5:	// Проверка Р2-30 и Р3-06
	IF Asda.P2_30=5 AND Asda.P3_06=3 THEN
		CNT_0:=90;
	ELSE
		IF CNT_1 = 2 THEN					// Если безушпешные 3 попытки
			Asda.E_CODE.2:=1;				// Ошибка инициализации Р2-30 или Р3-06
		ELSE		
			// Запись Р2-30=5 и Р3-06=3
			AddWriteCmd (wCmd:=wcAsda_P5_30);	// См. фукнцию AddWriteCmd	
			AddWriteCmd (wCmd:=wcAsda_P3_06);	// См. фукнцию AddWriteCmd	
			CNT_0:=10;							// Переход
		END_IF
	END_IF

10:	// Выдержка времени 1 сек
	TM_LOC (IN:=TRUE, PT:=T#1S);
	IF TM_LOC.Q THEN
		TM_LOC (IN:=FALSE);				// Сброс таймера
		CNT_0:=20;						// Переход
	END_IF

20:	// Чтение Р2-30 и Р3-06
	AddReadCmd (rCmd:=rcAsda_P2_30);	// Чтение Р2-30
	AddReadCmd (rCmd:=rcAsda_P3_06);	// Чтение Р3-06
	CNT_0:=30;							// Переход

30:	// Выдержка времени 1 сек
	TM_LOC (IN:=TRUE, PT:=T#1S);
	IF TM_LOC.Q THEN
		TM_LOC (IN:=FALSE);				// Сброс таймера
		CNT_1:=CNT_1+1;					// Увеличиваем счётчик	
		CNT_0:=5;						// Переход на начальную проверку
	END_IF

90:	// Выдержка времени 2 сек
	TM_LOC (IN:=TRUE, PT:=T#2S);
	IF TM_LOC.Q THEN
		CNT_0:=100;
	END_IF

100: // Конец 
	Asda.IsInit:=TRUE;					// Установка флага инициализации
	TM_LOC (IN:=FALSE);
	TM_DOG (IN:=FALSE);
	RESULT:=TRUE;

END_CASE

// Обнаружение ошибок
BREAK:=Asda.E_CODE <> 0;
IF BREAK THEN
	CNT_0:=100;
END_IF
END_ACTION

ACTION ST_Error_entry:

// Сброс селектора
CNT_0:=0;

// Сброс тайтера
TM_LOC (IN:=FALSE, PT:=T#2S);

// Сброс флага
RESULT:=0;

// Установить флаг ожидания сброса ошибки
Asda.WAIT_ERR:=TRUE;
END_ACTION

ACTION ST_Wait_entry:

// Включим флаг ожидания 
Asda.WAIT:=TRUE;

// Индекс сообщения
Asda.text_id:=0;
END_ACTION

ACTION ST_Servo_On_active:
CASE CNT_0 OF
0:
	// Устанавливает сигнал СБРОС и SERVO_ON на сервоприводе
	Asda.text_id:=6;					// Индекс сообщения
	AddWriteCmd (wCmd:=wcAsda_P4_07_4);	// См. функцию AddWriteCmd
	CNT_0:=10;							// Переход

10:	// Задержка 3 сек
	TM_LOC (IN:=TRUE, PT:=T#3S);
	IF TM_LOC.Q THEN
		TM_LOC (IN:=FALSE);			// Сброс таймера
		CNT_0:=20;					// Переход
	END_IF

20:	// Сбрасываем сигнал СБРОС при включенном SERVO_ON
	AddWriteCmd (wCmd:=wcAsda_P4_07_2);	// См. функцию AddWriteCmd
	CNT_0:=30;							// Переход

30:	// Задержка 1 сек
	TM_LOC (IN:=TRUE, PT:=T#1S);
	IF TM_LOC.Q THEN
		TM_LOC (IN:=FALSE);			// Сброс таймера
		CNT_0:=100;					// Переход
	END_IF

100: // Конец
	Asda.IsServo_ON:=TRUE;
	RESULT:=TRUE;

END_CASE
END_ACTION

ACTION ST_Parking_active:

CASE CNT_0 OF
	
0:	// Сообщение о движении в реперную точку
	IF Asda.IsServo_ON THEN
		Asda.text_id:=11;					// Индекс сообщения
		AddWriteCmd (wCmd:=wcAsda_Parking);	// Запуск

		CNT_0:=10;
	ELSE
		CNT_0:=100;
	END_IF
	
10:	// Ожидание 1 сек пока Р5-07 станет отличным от 20013 (Выполняется программа: PR#13 - парковка
	TM_LOC (IN:=TRUE, PT:=T#1S);
	IF TM_LOC.Q THEN
		TM_LOC (IN:=FALSE);
		CNT_0:=20;
	END_IF

20: // Ждём пока значение Р5-07 станет равно 20013 - значение окончания HOMING
	IF Asda.P5_07 = 20013 THEN
		CNT_0:=100;
	END_IF

100: // Завершение
	TM_LOC (IN:=FALSE);
	TM_DOG (IN:=FALSE);
	RESULT:=TRUE;

END_CASE

// Обнаружение предупреждения WARN (концевики в основном)
IF Asda.P0_46.10 THEN
	Asda.E_CODE.1:=1;		// WARN ()
END_IF

// Обнаруживаем ошибку АВАРИЯ СЕРВОПРИВОДА 
IF Asda.P0_46.6 THEN
	Asda.E_CODE.0:=1;		// ALRM (Авария привода)
END_IF

// Сторожевой таймер
TM_DOG (IN:=TRUE, PT:=tm_parking);
IF TM_DOG.Q THEN
	Asda.E_CODE.3:=1;		// Превышено время операции Homing
END_IF

// Ошибку блокировки игнорируем, так как будем использовать парковку
// при обработке падения темпераруры (Asda.Block) в рабочем режиме
BREAK:=Asda.E_CODE <> 0;
IF BREAK THEN 
	CNT_0:=100;
END_IF
END_ACTION

ACTION ST_Cont_entry:


// Переходим на ожидание
IF OP = OP_END THEN
    PROC:=PR_WAIT;
END_IF;
END_ACTION

ACTION ST_Stop_active:

// Экстренный останов
CASE CNT_0 OF
	
0:	// Подаём сигнал экстренного СТОП
	AddWriteCmd (wCmd:=wcAsda_Stop); 
	CNT_0:=10;
	
10:	// Небольшая задержка
	TM_LOC (IN:=TRUE, PT:=T#1S);
	IF TM_LOC.Q THEN
		TM_LOC (IN:=FALSE);
		CNT_0:=100;
	END_IF

100: // Конец
	RESULT:=TRUE;	

END_CASE
END_ACTION

ACTION ST_PR_Init_active:
CASE CNT OF

0:	// Проверка нинциализации
	IF Asda.P2_30=5 AND Asda.P3_06=3 THEN
		OP:=OP_NO;
	ELSE
		OP:=OP_INIT;
	END_IF

	CNT:=10;

10:	// Установка параметров
	OP:=OP_PARAMS;
	CNT:=100;
	
100: // Конец
	OP:=OP_END;
	
END_CASE
END_ACTION

ACTION Init_entry:

// Сброс селектора
CNT:=0;

// Начальная процедура - ожидание
PROC:=PR_WAIT;

// Сброс операции
OP:=OP_NO;

Asda.IsHoming:=FALSE;
Asda.IsInit:=FALSE;
Asda.IsServo_ON:=FALSE;
Asda.Pusk:=FALSE;
//Asda.Block:=TRUE;
Asda.WAIT:=FALSE;
Asda.WAIT_ERR:=FALSE;
Asda.WAIT_WORK:=FALSE;
Asda.P2_30:=0;
Asda.P3_06:=0;
Asda.E_CODE:=0;
Asda.text_id:=12;	// Ожидание соединения

// Проверка сохраненной ранее структуры W_Period: TPeriod
IF NOT IsRegValid (ADR (REG_W)) THEN
	REG_W:=REG_DEF;
END_IF
END_ACTION

ACTION ST_OFF_active:

CASE CNT OF
	
0:	// Инициализация сервопривода
	OP:=OP_INIT;
	CNT:=10;

10:	// Отключение сервопривода 
	OP:=OP_SERVO_OFF;
	CNT:=20;
	
20:	// Конец
	OP:=OP_END;

END_CASE
END_ACTION

ACTION ST_Stop_entry:

// Сброс селектора
CNT_0:=0;

// Сброс таймера
TM_LOC (IN:=FALSE, PT:=T#2S);

// Сброс флага
RESULT:=FALSE;

// Индекс сообщения
Asda.text_id:=7;
END_ACTION

ACTION ST_Pulsing_active:
CASE CNT_0 OF
	
0: 	// Начало
	Asda.text_id:=3;			// Индекс сообщения
	Asda.WAIT_WORK:=TRUE;		// Флаг состояния работы
	CNT_0:=10;
	
10:	// Запись команды на пульсирование
	AddWriteCmd (wCmd:=wcAsda_Working);
	CNT_0:=20;			// Переход
	
20:	// Ждём 1 сек пока значение Р5-07 изменится
	TM_LOC (IN:=TRUE, PT:=T#1S);
	IF TM_LOC.Q THEN
		TM_LOC (IN:=FALSE);
		CNT_0:=30;
	END_IF

30:

	// ЗДЕСЬ ИДЁТ ОСНОВНАЯ РАБОТА
	
	IF NOT Asda.Pusk THEN
		// Выход при автоматическом режиме
		CNT_0:=100;
	END_IF

100: // Выход

	TM_LOC (IN:=FALSE);
	TM_DOG (IN:=FALSE);
	Asda.WAIT_WORK:=FALSE;		// Флаг состояния работы
	RESULT:=TRUE;

END_CASE

// Обнаружение ошибок
IF Asda.P0_46.10 THEN
	Asda.E_CODE.1:=1;		// WARN ()
END_IF

IF Asda.P0_46.6 THEN
	Asda.E_CODE.0:=1;		// ALRM (Авария привода)
END_IF

IF Asda.E_CODE <> 0 THEN
	BREAK:=TRUE;
END_IF
	
IF BREAK THEN
	CNT_0:=100;
END_IF
END_ACTION

ACTION ST_Wait_exit:

// Выключим флаг ожидания 
Asda.WAIT:=FALSE;

// Сброс селектора
CNT:=0;

// Сброс операции
OP:=OP_NO;
END_ACTION

ACTION ST_Empty_exit:
// Внутренний селектор
CNT_0:=0;
CNT_1:=0;

// Внутренние таймеры
TM_LOC (IN:=FALSE, PT:=T#1S);
TM_DOG (IN:=FALSE, PT:=T#1S);

// Сброс флага
RESULT:=FALSE;

// Сброс прерывания
BREAK:=FALSE;
END_ACTION

ACTION ST_Params_active:

CASE CNT_0 OF

0:	// Установка индекса сообщения параметров
	Asda.text_id:=9;
	CNT_0:=10;
	
10:	// Установка параметров сервопривода
	Asda.SelButton:=sbPeriod;		// Параметры периода Asda
	AsdaSetPeriod ();

	CNT_0:=90;

90:	// Выдержка времени 2 сек
	TM_LOC (IN:=TRUE, PT:=T#2S);
	IF TM_LOC.Q THEN
		CNT_0:=100;
	END_IF

100: // Конец 
	TM_LOC (IN:=FALSE);
	TM_DOG (IN:=FALSE);
	RESULT:=TRUE;
	
END_CASE
END_ACTION

ACTION ST_FIRST_active:
CASE CNT OF

0:	// Включение сервопривода (попутно с сбросом аварии)
	OP:=OP_SERVO_ON;
	CNT:=20;			// Переход 
	
20:	// Установка параметров
	OP:=OP_PARAMS;
	CNT:=30;
	
30:	// Homing
	OP:=OP_HOMING;
	CNT:=40;
	
40:	// Конец
	OP:=OP_END;

END_CASE
END_ACTION

ACTION ST_WORK_active:

CASE CNT OF
0:	// Включение пульсирования
	OP:=OP_PULSING;
	CNT:=10;

10:	// Возвращение в реперную точку
	OP:=OP_PARKING;
	CNT:=20;	
	
20:	// Конец
	OP:=OP_END;

	
END_CASE
END_ACTION

ACTION ST_Wait_active:


// Проверяемна наличие Connect
IF Asda.Connect THEN

	IF NOT Asda.IsInit THEN
		// Инициализация
		PROC:=PR_INIT;
		FIRST:=TRUE;
		RESULT:=TRUE;
		RETURN;
	END_IF

	// Ожидание снятия блокировки (при достижении температуры)		
	IF NOT Asda.Block THEN

		// Включаем сервопривод через Servo_ON
		IF NOT Asda.IsServo_ON THEN			
			PROC:=PR_FIRST;
			RESULT:=TRUE;

		ELSIF Asda.Pusk THEN
			PROC:=PR_WORK;
			RESULT:=TRUE;
		
		END_IF

	// Появление блокировки (при снижении температуры)
	ELSE
		// Отключаем сервопривод через Servo_OFF
		IF Asda.IsServo_ON THEN
			// Инициализация, затем отключение сервопривода 
			PROC:=PR_OFF;
			RESULT:=TRUE;
		END_IF

	END_IF
END_IF
END_ACTION

ACTION ST_RESET_active:
// Процедура сброса, например после ошибки

CASE CNT OF
	
0:	// Homing
	OP:=OP_HOMING;
	CNT:=10;

10:	// Конец
	OP:=OP_END;
	
END_CASE
END_ACTION

ACTION ST_Error_active:

CASE CNT_0 OF
0:	// Ожидаем появления сигнала "СБРОС АВАРИИ"

	Asda.text_id:=10;			// Обработка ошибки
	IF ALARM_RESET THEN
		CNT_0:=10;
	END_IF

10:	// Действуем в зависимости от возникшей ошибки
	// - сигнал ALRM
	IF Asda.E_CODE.0 THEN	
		PROC:=PR_AVAR;			//	Переход на обработку аварии 	

	// - сигнал WARN	
	ELSIF Asda.E_CODE.1 THEN
		PROC:=PR_RESET;			//	Переход на Homing 	

	// - Ошибка инициализации Р2-30 или Р3-06	
	ELSIF Asda.E_CODE.2 THEN
		PROC:=PR_FIRST;			// Переход на инициализацию		
	
	// - Превышено время операции HOMING	
	ELSIF Asda.E_CODE.3 THEN
		PROC:=PR_RESET;			// Переход на Homing
	
	// - Превышено время операции отладки	
	ELSIF Asda.E_CODE.5 THEN
		PROC:=PR_RESET;			// Переход на Homing
	
	// Тестовая ошибка
	ELSIF Asda.E_CODE.6 THEN
		PROC:=PR_WAIT;			// Переход на Ожидание

	// Неизвестная ошибка
	ELSE
		PROC:=PR_WAIT;
	END_IF
	
	CNT_0:=20;					// Переход на ожидание сброса аварии

20:	// Сброс аварии
	Asda.E_CODE:=0;
	CNT_0:=30;

30: // Ожидание пропадания сигнала SBROS_AVARII
	IF NOT ALARM_RESET THEN
		CNT_0:=100;
	END_IF

100: // Конец
	RESULT:=TRUE;

END_CASE
END_ACTION

ACTION ST_Error_exit:

// Сброс операции
OP:=OP_NO;

// Сброс главного селектора
CNT:=0;

// Сбросить флаг ожидания сброса ошибки
Asda.WAIT_ERR:=FALSE;
END_ACTION

END_PROGRAM

// Device/Application/SRC/AddWriteCmd
PROGRAM AddWriteCmd
VAR_INPUT
	wCmd	: TWriteCmd;
END_VAR

VAR
	WR_CMDS		: ARRAY [0..11] OF WORD:=[5, 3, 0, 1, 2, 3, 0, 10, 13, 1000, 14, 15];	// Слова для команд сервопривода
	CH_CMDS		: ARRAY [0..1] OF WORD:=[0, 1];
	CH_UST		: INT;

END_VAR

// В зависимости от команды ...
CASE wcmd OF
	
	//=====================================================================================
	// КОМАНДЫ ПЕРВОНАЧАЛЬНОЙ ИНИЦИАЛИЗАЦИИ
	//=====================================================================================
	wcAsda_P5_30	: QueuePushReg (ADR (COM1_PRG.WR_REGS), ADR_ASDA, 16#023C, ADR (WR_CMDS[0]), 1);	// Параметр  Р2-30 -> 5 (отключение записи в EEPROM) - 5 в старшем байте!
	wcAsda_P3_06	: QueuePushReg (ADR (COM1_PRG.WR_REGS), ADR_ASDA, 16#030C, ADR (WR_CMDS[1]), 1);	// Параметр  Р3-06 -> 3 (способ управления дискретными входами) - 3 в старшем байте!
	wcAsda_P4_07_1	: QueuePushReg (ADR (COM1_PRG.WR_REGS), ADR_ASDA, 16#040E, ADR (WR_CMDS[2]), 1);	// Запись 00 в Р4-07 (servo_off)
	wcAsda_P4_07_2	: QueuePushReg (ADR (COM1_PRG.WR_REGS), ADR_ASDA, 16#040E, ADR (WR_CMDS[3]), 1);	// Запись 01 в Р4-07 (servo_on)
	wcAsda_P4_07_3	: QueuePushReg (ADR (COM1_PRG.WR_REGS), ADR_ASDA, 16#040E, ADR (WR_CMDS[4]), 1);	// Запись 10 в Р4-07 (сброс ошибок и выключенние servo_off)
	wcAsda_P4_07_4	: QueuePushReg (ADR (COM1_PRG.WR_REGS), ADR_ASDA, 16#040E, ADR (WR_CMDS[5]), 1);	// Запись 11 в Р4-07 (сброс ошибок с включенным servo_on)	
	//=====================================================================================
	// КОМАНДЫ УПРАВЛЕНИЯ ASDA
	//=====================================================================================
	wcAsda_Homing	: QueuePushReg (ADR (COM1_PRG.WR_REGS), ADR_ASDA, 16#050E, ADR (WR_CMDS[6]), 1);	// Команда HOMING - запись в Р5-07 числа 0
	wcAsda_Working	: QueuePushReg (ADR (COM1_PRG.WR_REGS), ADR_ASDA, 16#050E, ADR (WR_CMDS[7]), 1);	// Команда WORKING - запись в Р5-07 числа 10
	wcAsda_Parking	: QueuePushReg (ADR (COM1_PRG.WR_REGS), ADR_ASDA, 16#050E, ADR (WR_CMDS[8]), 1);	// Команда PARKING - запись в Р5-07 числа 13
	wcAsda_Stop		: QueuePushReg (ADR (COM1_PRG.WR_REGS), ADR_ASDA, 16#050E, ADR (WR_CMDS[9]), 1);	// КОМАНДА "СТОП" - запись в Р5-07 числа 1000
	wcAsda_Forward	: QueuePushReg (ADR (COM1_PRG.WR_REGS), ADR_ASDA, 16#050E, ADR (WR_CMDS[10]), 1);	// Команда вперёд - запись в Р5-07 числа 14
	wcAsda_Backward	: QueuePushReg (ADR (COM1_PRG.WR_REGS), ADR_ASDA, 16#050E, ADR (WR_CMDS[11]), 1);	// Команда назад - запись в Р5-07 числа 15
	//=====================================================================================
	// КОМАНДЫ ЧИЛЛЕРА
	//=====================================================================================
	wcChiller_Ust:
		CH_UST :=REAL_TO_INT (REG_W.T_CHIL * 10.0);
		QueuePushReg (ADR (COM3_PRG.WR_REGS), ADR_CHILLER, 11, ADR (CH_UST), 1);						// Запись уставки Чиллера

	wcChiller_Start	: QueuePushReg (ADR (COM3_PRG.WR_REGS), ADR_CHILLER, 12, ADR (CH_CMDS[1]), 1);		// Старт Чиллера
	wcChiller_Stop	: QueuePushReg (ADR (COM3_PRG.WR_REGS), ADR_CHILLER, 12, ADR (CH_CMDS[0]), 1);		// Стоп Чиллера
	
END_CASE

END_PROGRAM

// Device/Application/SRC/AddReadCmd
PROGRAM AddReadCmd
VAR_INPUT
	rCmd	: TReadCmd;
END_VAR

VAR
END_VAR


// В зависимости от команды 
CASE rCmd OF
	//=====================================================================================
	// КОМАНДЫ ДЛЯ ПЕРВОНАЧАЛЬНОЙ ИНИЦИАЛИЗАЦИИ ASDA_A2
	//=====================================================================================
	rcAsda_P2_30	: QueuePushReg (ADR (COM1_PRG.RD_REGS), ADR_ASDA, 16#023C, ADR (Asda.P2_30), 1); 			// Чтение Р2-30 (отключение записи в EEPROM, д.б.= 5)
	rcAsda_P3_06	: QueuePushReg (ADR (COM1_PRG.RD_REGS), ADR_ASDA, 16#030C, ADR (Asda.P3_06), 1); 			// Чтение Р3-06 (способ управления дискретными входами, д.б.= 3)
	
	
END_CASE

END_PROGRAM

// Device/Application/SRC/IsRegValid
FUNCTION IsRegValid : BOOL
VAR_INPUT
	pr : POINTER TO TReg;
	
END_VAR
VAR
	I: INT;
END_VAR

IsRegValid:=FALSE;

// Температуры
// Проверка температур
FOR I:=0 TO NUM_TEMPS-1 DO
	IF (pr^.TEMPS[I] < 0) OR (pr^.TEMPS[I] > T_CRITICALS[I]) THEN
		RETURN;
	END_IF
END_FOR

// Температура чиллера
IF (pr^.T_CHIL < 0) OR (pr^.T_CHIL > T_CHIL_CRITICAL) THEN
	RETURN;
END_IF

// Частота колебаний
IF pr^.Freq < FREQ_MIN OR pr^.Freq > FREQ_MAX THEN
	RETURN;
END_IF 

// Смещение 1-го полупериода
IF pr^.Period.Offsets[0] < (REP_MM + 0.3) OR pr^.Period.Offsets[0] > (WORK_SIZE + REP_MM - 0.3) THEN
	RETURN;
END_IF

// Смещение 2-го полупериода
IF pr^.Period.Offsets[1] < (REP_MM + 0.3) OR pr^.Period.Offsets[1] > (WORK_SIZE + REP_MM - 0.3) THEN
	RETURN;
END_IF

// Проценты полупериодов
IF pr^.Period.Per_FirstHP < ASDA_HP_MIN OR pr^.Period.Per_FirstHP > ASDA_HP_MAX THEN
	RETURN;
END_IF

// Проценты импульсов
IF pr^.Period.Per_Pulses[0] < ASDA_PULSE_MIN OR pr^.Period.Per_Pulses[0] > ASDA_PULSE_MAX THEN
	RETURN;
END_IF

IF pr^.Period.Per_Pulses[1] < ASDA_PULSE_MIN OR pr^.Period.Per_Pulses[1] > ASDA_PULSE_MAX THEN
	RETURN;
END_IF

// Проценты уровня
IF pr^.Period.Per_Levels[0] < ASDA_LEVEL_MIN OR pr^.Period.Per_Levels[0] > ASDA_LEVEL_MAX THEN
	RETURN;
END_IF

IF pr^.Period.Per_Levels[1] < ASDA_LEVEL_MIN OR pr^.Period.Per_Levels[1] > ASDA_LEVEL_MAX THEN
	RETURN;
END_IF

// Скорость заготовки
IF pr^.Speed < SPEED_MIN OR pr^.Speed >= SPEED_MAX THEN
	RETURN;
END_IF

// Длина заготовки
IF pr^.Length < LEN_MIN OR pr^.Length > LEN_MAX THEN
	RETURN;
END_IF

// Производительность
IF pr^.Qm < QM_MIN OR pr^.Qm > QM_MAX THEN
	RETURN;
END_IF

IsRegValid:=TRUE;

END_FUNCTION

// Device/Application/SRC/AsdaSetPeriod
PROGRAM AsdaSetPeriod
VAR
	dRep		: DINT;
	wSpeeds		: ARRAY [0..1] OF WORD;			// обороты в мин
	wAccs		: ARRAY [0..3] OF WORD;			// обороты в мин
	wDels		: ARRAY [0..1] OF WORD;			// милисекунды
	dOffsets	: ARRAY [0..1] OF DINT;
	dist		: REAL;
	tPeriod		: REAL;			
	tHalfs		: ARRAY [0..1] OF REAL;
	tPulses		: ARRAY [0..1] OF REAL;
	tLevels		: ARRAY [0..1] OF REAL;
	tAccs		: ARRAY [0..1] OF REAL;
	midSpeeds	: ARRAY [0..1] OF REAL;
	vSpeeds		: ARRAY [0..1] OF REAL;
END_VAR


CASE Asda.SelButton OF

sbPeriod:	// УСТАНОВКА ПАРАМЕТРОВ ПЕРИОДА

	// 1. Сначала записать положение реперной точки P6-01, адрес 16х0602
	dRep:=REAL_TO_DINT (REP_MM * PUU_PER_MM);
	QueuePushReg (ADR (COM1_PRG.WR_REGS), ADR_ASDA, 16#0602, ADR (dRep), 2);			// Р6-01 Положение реперной точки

	// 2. Запись перемещения 1-го полупериода, т.к. оно используется при вычислении следующих параметров
	dOffsets[0]:=REAL_TO_DINT (REG_W.Period.Offsets[0] * PUU_PER_MM);
	QueuePushReg (ADR (COM1_PRG.WR_REGS), ADR_ASDA, 16#062A, ADR (dOffsets[0]), 2);	// Р6-21 Смещение 1-го полупериода рабочее
	QueuePushReg (ADR (COM1_PRG.WR_REGS), ADR_ASDA, 16#063A, ADR (dOffsets[0]), 2);	// Р6-29 Смещение 1-го полупериода для ШАГА позиционирования 14 (ручное перемещение)

	// Запись перемещения 2-го полупериода, т.к. оно используется при вычислении следующих параметров
	dOffsets[1]:=REAL_TO_DINT (REG_W.Period.Offsets[1] * PUU_PER_MM);
	QueuePushReg (ADR (COM1_PRG.WR_REGS), ADR_ASDA, 16#062E, ADR (dOffsets[1]), 2);	// Р6-23 Смещение 2-го полупериода
	QueuePushReg (ADR (COM1_PRG.WR_REGS), ADR_ASDA, 16#063E, ADR (dOffsets[1]), 2);	// Р6-31 Смещение 2-го полупериода для шага позиционирования 15 (ручное перемещение)

	// Время периода в секундах
	tPeriod:= 1 / REG_W.Freq;
	
	// Времена полупериодов в секундах
	tHalfs[0]:=tPeriod * REG_W.Period.Per_FirstHP / 100;
	tHalfs[1]:=tPeriod - tHalfs[0];
	
	// Времена импульсов в секундах
	tPulses[0]:=tHalfs[0] * REG_W.Period.Per_Pulses[0] / 100;
	tPulses[1]:=tHalfs[1] * REG_W.Period.Per_Pulses[1] / 100;
	
	// Фронты полупериодов (импульсов) в секундах - Длина импульса минус длина уровня, делённая на 2
	tAccs[0]:=tPulses[0] * (100 - REG_W.Period.Per_Levels[0]) / 200;
	tAccs[1]:=tPulses[1] * (100 - REG_W.Period.Per_Levels[1]) / 200;
	
	// Уровни полупериодов
	tLevels[0]:=tPulses[0] * REG_W.Period.Per_Levels[0] / 100;
	tLevels[1]:=tPulses[1] * REG_W.Period.Per_Levels[1] / 100;
	
	// Пройденный путь в мм
	dist:=ABS (REG_W.Period.Offsets[0] - REG_W.Period.Offsets[1]);
	
	// Средние скорости в мм/сек
	midSpeeds[0]:=dist / tPulses[0];
	midSpeeds[1]:=dist / tPulses[1];
	
	// Расчётные скорости в мм/сек
	vSpeeds[0]:=midSpeeds[0] * (2 * tAccs[0] + tLevels[0]) / (tAccs[0] + tLevels[0]);
	vSpeeds[1]:=midSpeeds[1] * (2 * tAccs[1] + tLevels[1]) / (tAccs[1] + tLevels[1]);
		
	// Пересчёт скорости, данные - l оборот => 5 мм перемещения
	// 5 мм/сек = 1 об/сек =>
	wSpeeds[0]:=REAL_TO_WORD (vSpeeds[0] * 60 * 10 / 5);	// Получили в об/мин (Нужно умножить на 10, т.к. в сервоприводе единица измерения скорости 0.1 об/мин)
	wSpeeds[1]:=REAL_TO_WORD (vSpeeds[1] * 60 * 10 / 5);	// Получили в об/мин

	// Пересчёт фронт и спада относительно скорости wSpeeds[0]
	wAccs[0]:=REAL_TO_WORD (tAccs[0] * 3000 * 1000 / wSpeeds[0]);	
	wAccs[1]:=REAL_TO_WORD (tAccs[0] * 3000 * 1000 / wSpeeds[0]);
	wAccs[2]:=REAL_TO_WORD (tAccs[1] * 3000 * 1000 / wSpeeds[1]);
	wAccs[3]:=REAL_TO_WORD (tAccs[1] * 3000 * 1000 / wSpeeds[1]);
	
	// Задержки в миллисекундах
	wDels[0]:=REAL_TO_WORD ((tHalfs[0] - tPulses[0]) * 1000.0);
	wDels[1]:=REAL_TO_WORD ((tHalfs[1] - tPulses[1]) * 1000.0);

	// Запись	
	QueuePushReg (ADR (COM1_PRG.WR_REGS), ADR_ASDA, 16#0528, ADR (wAccs[0]), 1);		// Р5-20 Фронт 1-го полупериода
	QueuePushReg (ADR (COM1_PRG.WR_REGS), ADR_ASDA, 16#052A, ADR (wAccs[1]), 1);		// Р5-21 Спад 1-го полупериода 
	QueuePushReg (ADR (COM1_PRG.WR_REGS), ADR_ASDA, 16#052C, ADR (wAccs[2]), 1);		// Р5-22 Фронт 2-го полупериода
	QueuePushReg (ADR (COM1_PRG.WR_REGS), ADR_ASDA, 16#052E, ADR (wAccs[3]), 1);		// Р5-23 Спад 2-го полупериода 

	QueuePushReg (ADR (COM1_PRG.WR_REGS), ADR_ASDA, 16#0578, ADR (wSpeeds[0]), 1);		// Р5-60 Скорость 1-го полупериода
	QueuePushReg (ADR (COM1_PRG.WR_REGS), ADR_ASDA, 16#057A, ADR (wSpeeds[1]), 1);		// Р5-61 Скорость 2-го полупериода 

	QueuePushReg (ADR (COM1_PRG.WR_REGS), ADR_ASDA, 16#0550, ADR (wDels[0]), 1);		// Р5-40 Задержка 1-го полупериода
	QueuePushReg (ADR (COM1_PRG.WR_REGS), ADR_ASDA, 16#0552, ADR (wDels[1]), 1);		// Р5-41 Задержка 2-го полупериода

// Команда Homing
sbHoming: AddWriteCmd (wCmd:=wcAsda_Homing);
	
// Движение вперёд
sbForward: AddWriteCmd (wCmd:=wcAsda_Forward);

// Движение назад
sbBackward: AddWriteCmd (wCmd:=wcAsda_Backward);

// Парковка
sbParking: AddWriteCmd (wCmd:=wcAsda_Parking);

// Работа (пульсирование)
sbWorking: AddWriteCmd (wCmd:=wcAsda_Working);
	
END_CASE

Asda.SelButton:=sbNo;
Asda.bCmd:=FALSE;

END_PROGRAM

// Device/Application/SRC_AUX/SWAP_BYTES
FUNCTION SWAP_BYTES : WORD
VAR_INPUT
	wValue : WORD;
END_VAR
VAR
END_VAR


SWAP_BYTES := SHL (wValue, 8) OR SHR (wValue, 8);

END_FUNCTION

// Device/Application/SRC/SET_FRAME_INDEX_EX
FUNCTION SET_FRAME_INDEX_EX : BYTE
VAR_INPUT
	Index : BYTE;
END_VAR
VAR
END_VAR
VAR // added by the converter: edge detectors and wires of the graphical bodies
    _w1 : ANY;
END_VAR

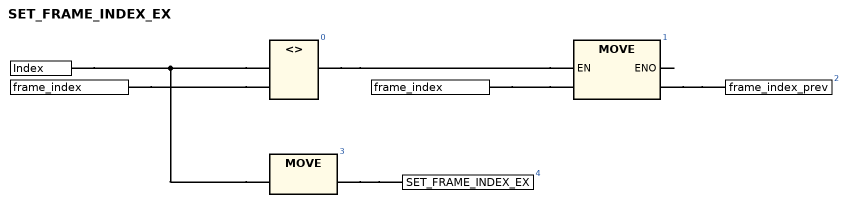
IF Index <> frame_index THEN _w1 := frame_index; END_IF
frame_index_prev := _w1;
SET_FRAME_INDEX_EX := Index;

END_FUNCTION

// Device/Application/SRC_AUX/BYTES_FROM_DINT
FUNCTION BYTES_FROM_DINT : BOOL
VAR_INPUT
	pBytes	: POINTER TO BYTE;
	iDint	: DINT;
END_VAR
VAR
	pB		: POINTER TO BYTE;
END_VAR

BYTES_FROM_DINT:=TRUE;

pB:=ADR(iDint);

pBytes[0]:=pB[1];
pBytes[1]:=pB[0];
pBytes[2]:=pB[3];
pBytes[3]:=pB[2];

END_FUNCTION

// Device/Application/SRC/MERGE_RGB
FUNCTION MERGE_RGB : DWORD
VAR_INPUT
	clR	: BYTE;
	clG	: BYTE;
	clB	: BYTE;
END_VAR
VAR
END_VAR

MERGE_RGB:=BYTE_TO_DWORD(255);
MERGE_RGB:=SHL(MERGE_RGB,8);
MERGE_RGB:=MERGE_RGB OR BYTE_TO_DWORD(clR);
MERGE_RGB:=SHL(MERGE_RGB,8);
MERGE_RGB:=MERGE_RGB OR BYTE_TO_DWORD(clG);
MERGE_RGB:=SHL(MERGE_RGB,8);
MERGE_RGB:=MERGE_RGB OR BYTE_TO_DWORD(clB);

END_FUNCTION

// Device/Application/SRC_FILE/WRITE_OPTIONS
FUNCTION WRITE_OPTIONS : BOOL
VAR_INPUT
	Show	: BOOL;
END_VAR
VAR
	hFile	: SysFile.RTS_IEC_HANDLE;	
	Result	: SysFile.RTS_IEC_RESULT;
	rSize	: __XWORD;
	wrBytes	: __XWORD;
	
END_VAR

WRITE_OPTIONS:=FALSE;
// Создаём новый файл
hFile:=SysFileOpen (OPTIONSFILE,SysFile.AM_WRITE, ADR (Result));
IF Result <> 0 THEN
	RETURN;
END_IF

rSize:=SIZEOF (TSetts);

wrBytes:=SysFileWrite(hFile, ADR (Setts), rSize, ADR (Result));
IF (Result=0) AND (wrBytes=rSize) THEN
	WRITE_OPTIONS:=TRUE;
END_IF

SysFileClose (hFile);

END_FUNCTION

// Device/Application/SRC_AUX/HiWord
FUNCTION HiWord : WORD
VAR_INPUT
	dValue	: DINT;
END_VAR	
VAR
	pW		: POINTER TO WORD;
END_VAR

pW:= ADR (dValue);
HiWord:=pW[1];

END_FUNCTION

// Device/Application/SRC_FILE/READ_OPTIONS
FUNCTION READ_OPTIONS : BOOL
VAR
	hFile	: SysFile.RTS_IEC_HANDLE;	
	Result	: SysFile.RTS_IEC_RESULT;
	fSize	: __XWORD;
	rSize	: __XWORD;
	rdBytes	: __XWORD;
	rdSetts	: TSetts;
	
END_VAR

READ_OPTIONS:=FALSE;

rSize:=SIZEOF(TSetts);

hFile:=SysFileOpen (OPTIONSFILE, SysFile.AM_READ, ADR (Result));
IF Result <> 0 THEN
	RETURN;
END_IF

//  Файл существует, проверяем размер файла
fSize:=SysFileGetSizeByHandle (hFile, ADR (Result));
IF Result <> 0 OR fSize <> rSize THEN
	SysFileClose(hFile);
	RETURN;	
END_IF

rdBytes:=SysFileRead(hFile, ADR (rdSetts), rSize, ADR (Result));	
IF Result = 0 AND rdBytes = rSize THEN
	Setts:=rdSetts;
	READ_OPTIONS:=TRUE;
END_IF

SysFileClose(hFile);

END_FUNCTION

// Device/Application/SRC_AUX/LoWord
FUNCTION LoWord : WORD
VAR_INPUT
	dValue	: DINT;
END_VAR
VAR
	pW		: POINTER TO WORD;
END_VAR

pW:= ADR (dValue);
LoWord:=pW[0];

END_FUNCTION

// Device/Application/SRC_AUX/LoByte
FUNCTION LoByte : BYTE
VAR_INPUT
	W	: WORD;
END_VAR
VAR
END_VAR

LoByte:=WORD_TO_BYTE (W AND 16#FF);

END_FUNCTION

// Device/Application/SRC_AUX/HiByte
FUNCTION HiByte : BYTE
VAR_INPUT
	W : WORD;
END_VAR
VAR
END_VAR

HiByte:= WORD_TO_BYTE (SHR (W, 8) AND 16#FF);

END_FUNCTION

// Device/Application/SRC_AUX/BYTES_FROM_INT
FUNCTION BYTES_FROM_INT : BOOL
VAR_INPUT
	pBytes	: POINTER TO BYTE;
	vInt	: INT;
END_VAR
VAR
	pB		: POINTER TO BYTE;
END_VAR

BYTES_FROM_INT:=TRUE;

pB:=ADR(vInt);
pBytes[0]:=pB[1];
pBytes[1]:=pB[0];

END_FUNCTION

// Device/Application/Visu/VIS_SETTS_2
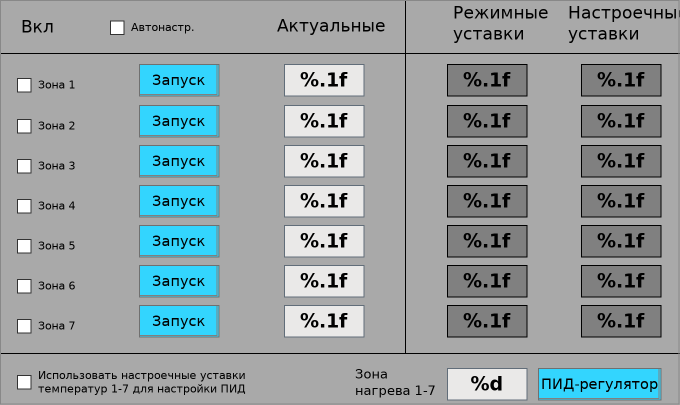
VISUALIZATION VIS_SETTS_2  // 680x405
    Checkbox (15,64 120x42), "Зона 1", variable: Nagrev.T_Enables.0
    Checkbox (15,105 120x42), "Зона 2", variable: Nagrev.T_Enables.1
    Checkbox (15,145 120x42), "Зона 3", variable: Nagrev.T_Enables.2
    Checkbox (15,185 120x42), "Зона 4", variable: Nagrev.T_Enables.3
    Checkbox (15,225 120x42), "Зона 5", variable: Nagrev.T_Enables.4
    Checkbox (15,265 120x42), "Зона 6", variable: Nagrev.T_Enables.5
    Checkbox (15,305 120x42), "Зона 7", variable: Nagrev.T_Enables.6
    Label (18,15 63x24), "Вкл"
    Button (139,64 80x32), "Запуск", colour toggle: Nagrev.Auto_IN.0, input disabled if: NOT AutoPIDActivate
        OnMouseClick: execute { Nagrev.Auto_OUT.0:=TRUE; }
    Button (139,105 80x32), "Запуск", colour toggle: Nagrev.Auto_IN.1, input disabled if: NOT AutoPIDActivate
        OnMouseClick: execute { Nagrev.Auto_OUT.1:=TRUE; }
    Button (139,145 80x32), "Запуск", colour toggle: Nagrev.Auto_IN.2, input disabled if: NOT AutoPIDActivate
        OnMouseClick: execute { Nagrev.Auto_OUT.2:=TRUE; }
    Button (139,185 80x32), "Запуск", colour toggle: Nagrev.Auto_IN.3, input disabled if: NOT AutoPIDActivate
        OnMouseClick: execute { Nagrev.Auto_OUT.3:=TRUE; }
    Button (139,225 80x32), "Запуск", colour toggle: Nagrev.Auto_IN.4, input disabled if: NOT AutoPIDActivate
        OnMouseClick: execute { Nagrev.Auto_OUT.4:=TRUE; }
    Button (139,265 80x32), "Запуск", colour toggle: Nagrev.Auto_IN.5, input disabled if: NOT AutoPIDActivate
        OnMouseClick: execute { Nagrev.Auto_OUT.5:=TRUE; }
    Button (139,305 80x32), "Запуск", colour toggle: Nagrev.Auto_IN.6, input disabled if: NOT AutoPIDActivate
        OnMouseClick: execute { Nagrev.Auto_OUT.6:=TRUE; }
    Checkbox (15,361 312x42), "Использовать настроечные уставки температур 1-7 для настройки ПИД", variable: zd_selector
    RoundedRectangle (447,64 80x32), "%.1f", text variable: REG_W.TEMPS[0], colour toggle: NOT zd_selector
    RoundedRectangle (447,105 80x32), "%.1f", text variable: REG_W.TEMPS[1], colour toggle: NOT zd_selector
    RoundedRectangle (447,145 80x32), "%.1f", text variable: REG_W.TEMPS[2], colour toggle: NOT zd_selector
    RoundedRectangle (447,185 80x32), "%.1f", text variable: REG_W.TEMPS[3], colour toggle: NOT zd_selector
    RoundedRectangle (447,225 80x32), "%.1f", text variable: REG_W.TEMPS[4], colour toggle: NOT zd_selector
    RoundedRectangle (447,265 80x32), "%.1f", text variable: REG_W.TEMPS[5], colour toggle: NOT zd_selector
    RoundedRectangle (447,305 80x32), "%.1f", text variable: REG_W.TEMPS[6], colour toggle: NOT zd_selector
    Label (450,1 107x49), "Режимные уставки"
    RoundedRectangle (581,64 80x32), "%.1f", text variable: zd_temps[0], colour toggle: zd_selector
        OnMouseClick: write the text variable via VisuDialogs.Numpad, min T_MINS_ZAD[6], max T_MAXS_ZAD[6], title "ТЕМПЕРАТУРА 7 ЗОНЫ"
    RoundedRectangle (581,105 80x32), "%.1f", text variable: zd_temps[1], colour toggle: zd_selector
        OnMouseClick: write the text variable via VisuDialogs.Numpad, min T_MINS_ZAD[0], max T_MAXS_ZAD[0]
    RoundedRectangle (581,145 80x32), "%.1f", text variable: zd_temps[2], colour toggle: zd_selector
        OnMouseClick: write the text variable via VisuDialogs.Numpad, min T_MINS_ZAD[0], max T_MAXS_ZAD[0]
    RoundedRectangle (581,185 80x32), "%.1f", text variable: zd_temps[3], colour toggle: zd_selector
        OnMouseClick: write the text variable via VisuDialogs.Numpad, min T_MINS_ZAD[0], max T_MAXS_ZAD[0]
    RoundedRectangle (581,225 80x32), "%.1f", text variable: zd_temps[4], colour toggle: zd_selector
        OnMouseClick: write the text variable via VisuDialogs.Numpad, min T_MINS_ZAD[0], max T_MAXS_ZAD[0]
    RoundedRectangle (581,265 80x32), "%.1f", text variable: zd_temps[5], colour toggle: zd_selector
        OnMouseClick: write the text variable via VisuDialogs.Numpad, min T_MINS_ZAD[0], max T_MAXS_ZAD[0]
    RoundedRectangle (581,305 80x32), "%.1f", text variable: zd_temps[6], colour toggle: zd_selector
        OnMouseClick: write the text variable via VisuDialogs.Numpad, min T_MINS_ZAD[0], max T_MAXS_ZAD[0]
    Label (565,1 127x47), "Настроечные уставки"
    RoundedRectangle (284,64 80x32), "%.1f", text variable: Nagrev.T_Actuals[0], colour variable: Nagrev.FillColors[0]
        p3450524324: Nagrev.FrameColors[0]
    RoundedRectangle (284,105 80x32), "%.1f", text variable: Nagrev.T_Actuals[1], colour variable: Nagrev.FillColors[1]
        p3450524324: Nagrev.FrameColors[1]
    RoundedRectangle (284,145 80x32), "%.1f", text variable: Nagrev.T_Actuals[2], colour variable: Nagrev.FillColors[2]
        p3450524324: Nagrev.FrameColors[2]
    RoundedRectangle (284,185 80x32), "%.1f", text variable: Nagrev.T_Actuals[3], colour variable: Nagrev.FillColors[3]
        p3450524324: Nagrev.FrameColors[3]
    RoundedRectangle (284,225 80x32), "%.1f", text variable: Nagrev.T_Actuals[4], colour variable: Nagrev.FillColors[4]
        p3450524324: Nagrev.FrameColors[4]
    RoundedRectangle (284,265 80x32), "%.1f", text variable: Nagrev.T_Actuals[5], colour variable: Nagrev.FillColors[5]
        p3450524324: Nagrev.FrameColors[5]
    RoundedRectangle (284,305 80x32), "%.1f", text variable: Nagrev.T_Actuals[6], colour variable: Nagrev.FillColors[6]
        p3450524324: Nagrev.FrameColors[6]
    Label (274,14 123x32), "Актуальные"
    Label (352,365 91x40), "Зона нагрева 1-7"
    Button (538,368 123x32), "ПИД-регулятор"
        OnMouseClick:  Dialog=DlgPids, Parameters={bDialogVar: b_dialog}, Selected={1: }, OpenModal=True, OpenCentered=True
    RoundedRectangle (447,368 80x32), "%d", text variable: Dvp.zone_index
        OnMouseClick: write the text variable via VisuDialogs.Numpad, min 1, max 7, title "Введите зону нагрева 1-7"
    Line (405,0) (405,353)
    Line (0,353) (680,353)
    Checkbox (108,9 140x37), "Автонастр.", variable: AutoPIDActivate
    Line (0,53) (680,53)
END_VISUALIZATION

// Device/Application/Visu/Main_Panel
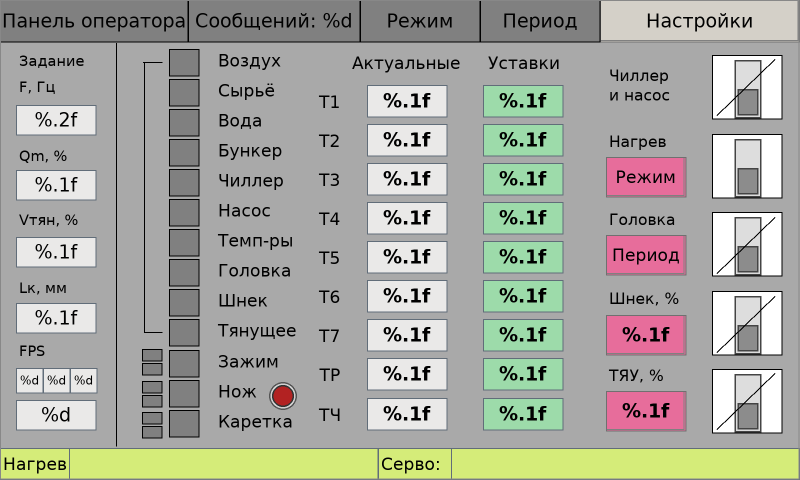
VISUALIZATION Main_Panel  // 800x480
    Rectangle (0,448 80x32), "Нагрев:"
    Frame (118,43 692x442), frame switch variable: frame_index
        shows VIS_OPERATOR()
        shows VIS_MSGS()
        shows VIS_REG()
        shows VIS_PERIOD()
        shows VIS_REG()
    Label (16,77 48x25), "F, Гц"
    RoundedRectangle (16,170 80x30), "%.1f", text variable: Shnek.Qm
    Label (16,146 77x27), "Qm, %"
    Label (16,210 92x26), "Vтян, %"
    RoundedRectangle (16,237 80x30), "%.1f", text variable: Pulling.Speed
    Label (16,278 59x25), "Lк, мм"
    RoundedRectangle (16,303 80x30), "%.1f", text variable: REG_W.Length
    RoundedRectangle (16,105 80x30), "%.2f", text variable: REG_W.Freq
    Label (16,51 79x20), "Задание"
    Line (116,43) (116,446)
    Rectangle (0,0 188x42), "Панель оператора", colour toggle: frame_index=0
        OnMouseClick: execute { SET_FRAME_INDEX (0); }
    Rectangle (188,0 172x42), "Сообщений: %d", text variable: alarm_count, colour toggle: frame_index=1
        OnMouseClick: execute { SET_FRAME_INDEX (1); }
    Button (600,0 200x42), "Настройки"
        OnMouseClick:  Assign=Setts_Panel, Type=Assignment
    Rectangle (69,448 309x32), text list: 'DvpTextList', text index: Nagrev.text_id
    Rectangle (378,448 80x32), "Серво:"
    Rectangle (451,448 349x32), text list: 'AsdaTextList', text index: Asda.text_id
    RoundedRectangle (16,400 80x30), "%d", text variable: FPS_FULL
    Label (16,341 59x25), "FPS"
    RoundedRectangle (16,368 27x25), "%d", text variable: COM1_PRG.FPS
    RoundedRectangle (43,368 27x25), "%d", text variable: COM2_PRG.FPS
    RoundedRectangle (70,368 27x25), "%d", text variable: COM3_PRG.FPS
    Rectangle (360,0 120x42), "Режим", colour toggle: frame_index=2
        OnMouseClick: execute { SET_FRAME_INDEX (2); }
    Rectangle (480,0 120x42), "Период", colour toggle: frame_index=3
        OnMouseClick: execute { SET_FRAME_INDEX (3); }
END_VISUALIZATION

// Device/Application/Visu/DlgConfirm
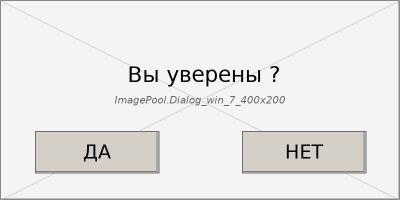
VISUALIZATION DlgConfirm  // 400x200
VAR_IN_OUT
	bDialogVar	: BOOL;
END_VAR
    Image (0,0 400x200), image: ImagePool.Dialog_win_7_400x200
    Button (35,131 124x42), "ДА"
        OnMouseClick:  Dialog=DlgConfirm, Result=OK, NumpadKeypadSet=True
        OnMouseClick: execute { bDialogVar:=TRUE; }
    Button (242,131 124x42), "НЕТ"
        OnMouseClick:  Dialog=DlgConfirm, Result=Cancel, NumpadKeypadSet=True
    Label (80,55 248x39), "Вы уверены ?"
END_VISUALIZATION

// Device/Application/Visu/Panel_Reg
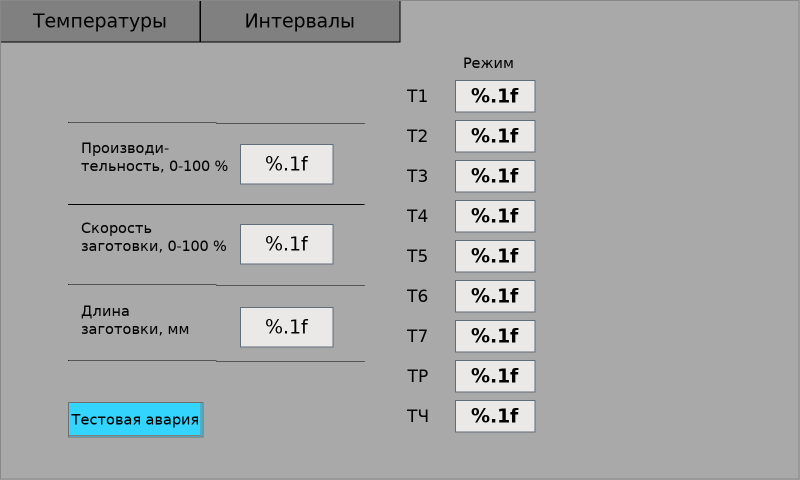
VISUALIZATION Panel_Reg  // 800x480
    Frame (6,47 734x398), frame switch variable: frame_index_reg
        shows VIS_REG()
        shows VIS_PERIOD()
    Rectangle (0,0 200x42), "Температуры", colour toggle: frame_index_reg=0
        OnMouseClick: execute { frame_index_reg:=0; }
    Rectangle (200,0 200x42), "Интервалы", colour toggle: frame_index_reg=1
        OnMouseClick: execute { frame_index_reg:=1; }
END_VISUALIZATION

// Device/Application/Visu/VIS_MSGS
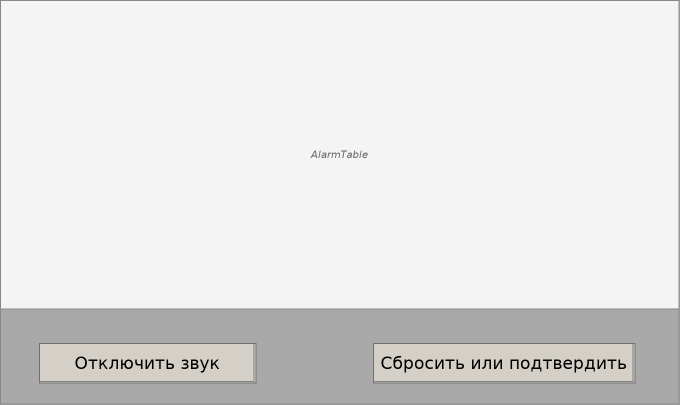
VISUALIZATION VIS_MSGS  // 680x405
VAR_IN_OUT
END_VAR
VAR
	bAckSel : BOOL;
	bAckVisible : BOOL;
	bHistory : BOOL;
	bFreezeScrlPos : BOOL;
END_VAR
    AlarmTable (0,0 679x309)
        Column[0]: ColumnTitle=Изоб
        Column[1]: ColumnTitle=Сообщение
        p1521930926: __All
        p1663851261: __All
        p428520879: bAckSel
        p2607059081: bAckVisible
        p3266827225: bHistory
        p3894972949: bFreezeScrlPos
    Button (39,343 217x40), "Отключить звук", colour toggle: ALARM_ZVUK AND NOT Setts.otkl_alarm_zvuk
        OnMouseClick: execute { ALARM_ZVUK:=FALSE; }
    Button (373,343 262x40), "Сбросить или подтвердить", colour toggle: ALARM_RESET
        toggle bAckVisible
        OnMouseClick: execute { ALARM_RESET:=TRUE; }
END_VISUALIZATION

// Device/Application/Visu/Setts_Panel
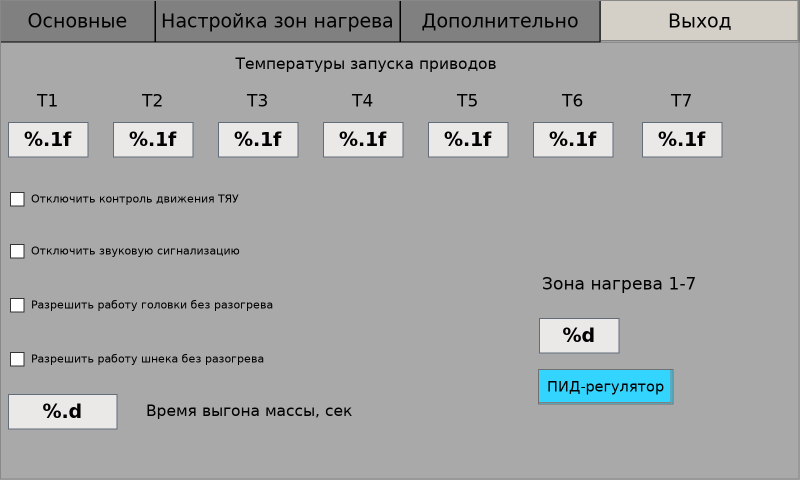
VISUALIZATION Setts_Panel  // 800x480
    Button (600,0 200x42), "Выход"
        OnMouseClick:  Assign=Main_Panel, Type=Assignment
    Rectangle (0,0 155x42), "Основные", colour toggle: frame_index_setts=0
        OnMouseClick: execute { frame_index_setts:=0; }
    Rectangle (155,0 245x42), "Настройка зон нагрева", colour toggle: frame_index_setts=1
        OnMouseClick: execute { frame_index_setts:=1; }
    Frame (0,43 793x430), frame switch variable: frame_index_setts
        shows VIS_SETTS_1()
        shows VIS_SETTS_2()
        shows VIS_SETTS_3()
    Rectangle (400,0 200x42), "Дополнительно", colour toggle: frame_index_setts=2
        OnMouseClick: execute { frame_index_setts:=2; }
END_VISUALIZATION

// Device/Application/Visu/VIS_REG
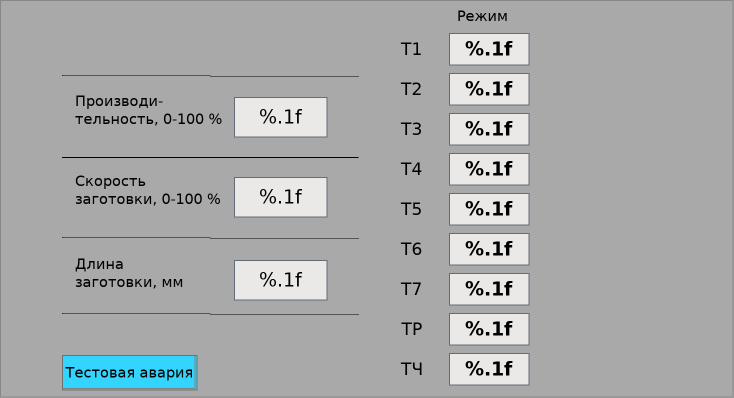
VISUALIZATION VIS_REG  // 734x398
    Line (62,313) (358,314)
    Line (62,237) (358,238)
    Line (62,157) (358,157)
    Line (62,75) (358,76)
    Label (72,91 162x53), "Производи- тельность, 0-100 %"
    Label (72,171 167x50), "Скорость заготовки, 0-100 %"
    RoundedRectangle (234,177 93x40), "%.1f", text variable: REG_W.Speed
        OnMouseClick: write the text variable via VisuDialogs.Numpad, min SPEED_MIN, max SPEED_MAX, title "Скорость заготовки, мм/сек"
    Label (72,254 126x53), "Длина заготовки, мм"
    RoundedRectangle (234,260 93x40), "%.1f", text variable: REG_W.Length
        OnMouseClick: write the text variable via VisuDialogs.Numpad, min LEN_MIN, max LEN_MAX, title "Длина заготовки, мм"
    RoundedRectangle (449,33 80x32), "%.1f", text variable: REG_W.TEMPS[0]
        OnMouseClick: write the text variable via VisuDialogs.Numpad, min T_MINS_ZAD[0], max T_MAXS_ZAD[0], title "ТЕМПЕРАТУРА 1 ЗОНЫ"
    Label (392,33 40x32), "T1"
    RoundedRectangle (449,73 80x32), "%.1f", text variable: REG_W.TEMPS[1]
        OnMouseClick: write the text variable via VisuDialogs.Numpad, min T_MINS_ZAD[1], max T_MAXS_ZAD[1], title "ТЕМПЕРАТУРА 2 ЗОНЫ"
    Label (392,73 40x32), "T2"
    RoundedRectangle (449,113 80x32), "%.1f", text variable: REG_W.TEMPS[2]
        OnMouseClick: write the text variable via VisuDialogs.Numpad, min T_MINS_ZAD[2], max T_MAXS_ZAD[2], title "ТЕМПЕРАТУРА3 ЗОНЫ"
    Label (392,113 40x32), "T3"
    RoundedRectangle (449,153 80x32), "%.1f", text variable: REG_W.TEMPS[3]
        OnMouseClick: write the text variable via VisuDialogs.Numpad, min T_MINS_ZAD[3], max T_MAXS_ZAD[3], title "ТЕМПЕРАТУРА 4 ЗОНЫ"
    Label (392,153 40x32), "T4"
    RoundedRectangle (449,193 80x32), "%.1f", text variable: REG_W.TEMPS[4]
        OnMouseClick: write the text variable via VisuDialogs.Numpad, min T_MINS_ZAD[4], max T_MAXS_ZAD[4], title "ТЕМПЕРАТУРА 5 ЗОНЫ"
    Label (392,193 40x32), "T5"
    RoundedRectangle (449,233 80x32), "%.1f", text variable: REG_W.TEMPS[5]
        OnMouseClick: write the text variable via VisuDialogs.Numpad, min T_MINS_ZAD[5], max T_MAXS_ZAD[5], title "ТЕМПЕРАТУРА 6 ЗОНЫ"
    Label (392,233 40x32), "T6"
    RoundedRectangle (449,273 80x32), "%.1f", text variable: REG_W.TEMPS[6]
        OnMouseClick: write the text variable via VisuDialogs.Numpad, min T_MINS_ZAD[6], max T_MAXS_ZAD[6], title "ТЕМПЕРАТУРА 7 ЗОНЫ"
    Label (392,273 40x32), "T7"
    RoundedRectangle (449,313 80x32), "%.1f", text variable: REG_W.TEMPS[7]
        OnMouseClick: write the text variable via VisuDialogs.Numpad, min T_MINS_ZAD[7], max T_MAXS_ZAD[7], title "ТЕМПЕРАТУРА РАСПЛАВА"
    Label (392,313 40x32), "TР"
    RoundedRectangle (449,353 80x32), "%.1f", text variable: REG_W.T_CHIL
        OnMouseClick: write the text variable via VisuDialogs.Numpad, min T_MIN_CHIL_ZAD, max T_MAX_CHIL_ZAD, title "ТЕМПЕРАТУРА ЧИЛЛЕРА"
    Label (392,353 40x32), "TЧ"
    Label (454,1 76x30), "Режим"
    RoundedRectangle (234,97 93x40), "%.1f", text variable: REG_W.Qm
        OnMouseClick: write the text variable via VisuDialogs.Numpad, min QM_MIN, max QM_MAX, title "Производительность, %"
    Button (62,355 135x35), "Тестовая авария"
        OnMouseClick: execute { ALARM_TEST:=TRUE; }
END_VISUALIZATION

// Device/Application/Visu/VIS_PERIOD
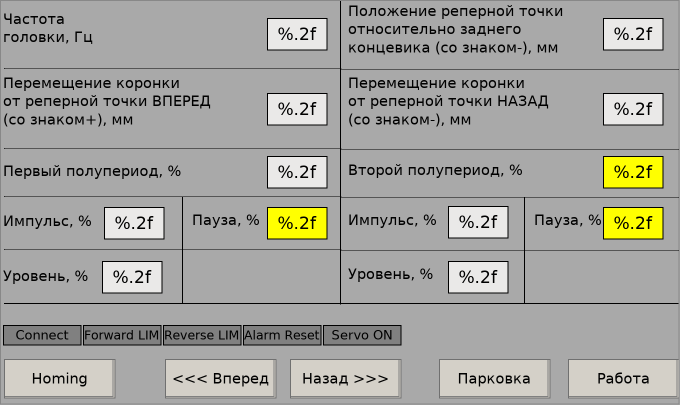
VISUALIZATION VIS_PERIOD  // 680x405
    RoundedRectangle (603,18 60x32), "%.2f", text variable: REP_MM
        OnMouseClick: write the text variable via VisuDialogs.Numpad, min REP_MIN, max REP_MAX, title "ЗАДАТЬ РЕПЕРНУЮ ТОЧКУ"
        OnDialogClosed: execute { Asda.SelButton:=sbPeriod; AsdaSetPeriod (); }
    Button (439,359 111x39), "Парковка", input disabled if: NOT Asda.WAIT
        OnMouseClick:  Dialog=DlgConfirm, Parameters={bDialogVar: Asda.bCmd}, Selected={1: }, OpenModal=True, OpenCentered=True
        OnDialogClosed: execute {
            IF Asda.bCmd THEN
            	Asda.SelButton:=sbParking;
            	AsdaSetPeriod ();
            END_IF
        }
    Label (345,1 220x69), "Положение реперной точки относительно заднего концевика (со знаком-), мм"
    Label (0,266 102x25), "Уровень, %"
    RoundedRectangle (102,261 60x32), "%.2f", text variable: REG_W.Period.Per_Levels[0]
        OnMouseClick: write the text variable via VisuDialogs.Numpad, min ASDA_LEVEL_MIN, max ASDA_LEVEL_MAX, title "УРОВЕНЬ ПЕРВОГО П/П"
        OnDialogClosed: execute { Asda.SelButton:=sbPeriod; AsdaSetPeriod (); }
    RoundedRectangle (448,261 60x32), "%.2f", text variable: REG_W.Period.Per_Levels[1]
        OnMouseClick: write the text variable via VisuDialogs.Numpad, min ASDA_LEVEL_MIN, max ASDA_LEVEL_MAX, title "УРОВЕНЬ ВТОРОГО П/П"
        OnDialogClosed: execute { Asda.SelButton:=sbPeriod; AsdaSetPeriod (); }
    Label (0,73 251x72), "Перемещение коронки от реперной точки ВПЕРЕД (со знаком+), мм"
    RoundedRectangle (267,93 60x32), "%.2f", text variable: REG_W.Period.Offsets[0]
        OnMouseClick: write the text variable via VisuDialogs.Numpad, min REP_MM + 0.3, max WORK_SIZE + REP_MM - 0.3, title "ПЕРЕМЕЩЕНИЕ 1-ГО П/П"
        OnDialogClosed: execute { Asda.SelButton:=sbPeriod; AsdaSetPeriod (); }
    Label (345,73 233x71), "Перемещение коронки от реперной точки НАЗАД (со знаком-), мм"
    RoundedRectangle (603,93 60x32), "%.2f", text variable: REG_W.Period.Offsets[1]
        OnMouseClick: write the text variable via VisuDialogs.Numpad, min REP_MM + 0.3, max WORK_SIZE + REP_MM - 0.3, title "ПЕРЕМЕЩЕНИЕ 2-ГО П/П"
        OnDialogClosed: execute { Asda.SelButton:=sbPeriod; AsdaSetPeriod (); }
    Button (568,359 111x39), "Работа", input disabled if: NOT Asda.WAIT
        OnMouseClick:  Dialog=DlgConfirm, Parameters={bDialogVar: Asda.bCmd}, Selected={1: }, OpenModal=True, OpenCentered=True
        OnDialogClosed: execute {
            IF Asda.bCmd THEN
            	Asda.SelButton:=sbWorking;
            	AsdaSetPeriod ();
            END_IF
        }
    Button (4,359 111x39), "Homing", input disabled if: NOT Asda.WAIT
        OnMouseClick:  Dialog=DlgConfirm, Parameters={bDialogVar: Asda.bCmd}, Selected={1: }, OpenModal=True, OpenCentered=True
        OnDialogClosed: execute {
            IF Asda.bCmd THEN
            	Asda.SelButton:=sbHoming;
            	AsdaSetPeriod ();
            END_IF
        }
    Button (165,359 111x39), "<<< Вперед", input disabled if: NOT Asda.WAIT
        OnMouseClick:  Dialog=DlgConfirm, Parameters={bDialogVar: Asda.bCmd}, Selected={1: }, OpenModal=True, OpenCentered=True
        OnDialogClosed: execute {
            IF Asda.bCmd THEN
            	Asda.SelButton:=sbForward;
            	AsdaSetPeriod ();
            END_IF
        }
    Button (290,359 111x39), "Назад >>>", input disabled if: NOT Asda.WAIT
        OnMouseClick:  Dialog=DlgConfirm, Parameters={bDialogVar: Asda.bCmd}, Selected={1: }, OpenModal=True, OpenCentered=True
        OnDialogClosed: execute {
            IF Asda.bCmd THEN
            	Asda.SelButton:=sbBackward;
            	AsdaSetPeriod ();
            END_IF
        }
    Line (4,68) (678,69)
    Line (4,303) (678,303)
    Line (4,196) (678,197)
    Label (0,161 214x23), "Первый полупериод, %"
    Label (345,160 216x23), "Второй полупериод, %"
    Label (345,264 97x25), "Уровень, %"
    Line (340,0) (340,304)
    RoundedRectangle (267,156 60x32), "%.2f", text variable: REG_W.Period.Per_FirstHP
        OnMouseClick: write the text variable via VisuDialogs.Numpad, min ASDA_HP_MIN, max ASDA_HP_MAX, title "ПЕРВЫЙ ПОЛУПЕРИОД"
        OnDialogClosed: execute { Asda.SelButton:=sbPeriod; AsdaSetPeriod (); }
    RoundedRectangle (603,156 60x32), "%.2f", text variable: 100 - REG_W.Period.Per_FirstHP
    Line (4,249) (678,250)
    Line (182,197) (182,303)
    RoundedRectangle (104,207 60x32), "%.2f", text variable: REG_W.Period.Per_Pulses[0]
        OnMouseClick: write the text variable via VisuDialogs.Numpad, min ASDA_PULSE_MIN, max ASDA_PULSE_MAX, title "ПЕРВЫЙ ПОЛУПЕРИОД"
        OnDialogClosed: execute { Asda.SelButton:=sbPeriod; AsdaSetPeriod (); }
    Label (0,211 94x23), "Импульс, %"
    Label (189,210 94x23), "Пауза, %"
    RoundedRectangle (267,207 60x32), "%.2f", text variable: 100-REG_W.Period.Per_Pulses[0]
    Label (345,210 94x23), "Импульс, %"
    RoundedRectangle (448,206 60x32), "%.2f", text variable: REG_W.Period.Per_Pulses[1]
        OnMouseClick: write the text variable via VisuDialogs.Numpad, min ASDA_PULSE_MIN, max ASDA_PULSE_MAX, title "ПЕРВЫЙ ПОЛУПЕРИОД"
        OnDialogClosed: execute { Asda.SelButton:=sbPeriod; AsdaSetPeriod (); }
    Label (531,210 94x23), "Пауза, %"
    RoundedRectangle (603,207 60x32), "%.2f", text variable: 100-REG_W.Period.Per_Pulses[1]
    Line (524,197) (524,303)
    Line (4,148) (678,149)
    RoundedRectangle (3,325 78x20), "Connect", colour toggle: Asda.Connect
    RoundedRectangle (243,325 78x20), "Alarm Reset", colour toggle: Asda.P4_07.1
    RoundedRectangle (323,325 78x20), "Servo ON", colour toggle: Asda.P4_07.0
    RoundedRectangle (163,325 78x20), "Reverse LIM", colour toggle: Asda.P4_07.2
    RoundedRectangle (83,325 78x20), "Forward LIM", colour toggle: Asda.P4_07.3
    Label (0,9 144x54), "Частота головки, Гц"
    RoundedRectangle (267,18 60x32), "%.2f", text variable: REG_W.Freq
        OnMouseClick: write the text variable via VisuDialogs.Numpad, min FREQ_MIN, max FREQ_MAX, title "ЧАСТОТА ГОЛОВКИ, Гц"
        OnDialogClosed: execute {
            //VisuDialogs.Numpad_VISU_STRUCT.bInit
            Asda.SelButton:=sbPeriod;
            AsdaSetPeriod ();
        }
END_VISUALIZATION

// Device/Application/Visu/VIS_OPERATOR
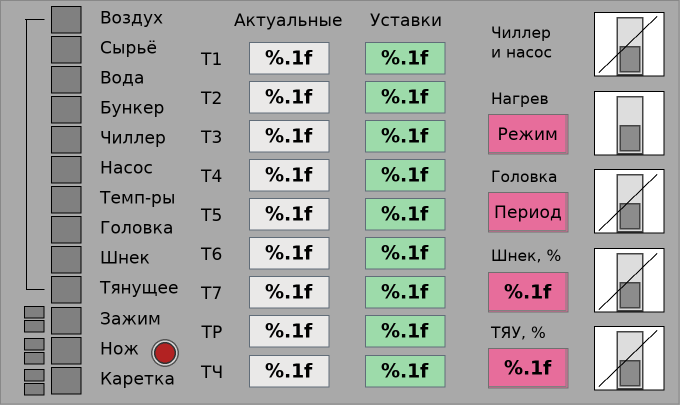
VISUALIZATION VIS_OPERATOR  // 680x405
    RoundedRectangle (594,91 70x64), colour variable: Nagrev.NagrevFillColor
        p3450524324: Nagrev.NagrevFrameColor
    DipSwitch (601,96 58x58), variable: Nagrev.Nagrev_on, behaviour: TOGGLE, style: Switch-DipSwitch-Gray
    RoundedRectangle (594,326 70x64), colour variable: Pulling.BtnFillColor
        p3450524324: Pulling.BtnFrameColor
    DipSwitch (601,331 58x58), variable: Pulling.Pusk, input disabled if: Pulling.Block, behaviour: TOGGLE, style: Switch-DipSwitch-Gray
    RoundedRectangle (594,248 70x64), colour variable: Shnek.FillColor
        p3450524324: Shnek.FrameColor
    DipSwitch (601,253 58x58), variable: Shnek.Pusk, input disabled if: Shnek.Block, behaviour: TOGGLE, style: Switch-DipSwitch-Gray
    RoundedRectangle (594,169 70x64), colour variable: Asda.BtnFillColor
        p3450524324: Asda.BtnFrameColor
    DipSwitch (601,174 58x58), variable: Asda.Pusk, input disabled if: Asda.Block, behaviour: TOGGLE, style: Switch-DipSwitch-Gray
    RoundedRectangle (249,42 80x32), "%.1f", text variable: Nagrev.T_Actuals[0], colour variable: Nagrev.FillColors[0]
        p3450524324: Nagrev.FrameColors[0]
    Label (192,43 40x32), "T1"
    RoundedRectangle (365,42 80x32), "%.1f", text variable: TEMPERS[0], colour toggle: Nagrev.Auto_IN.0
    RoundedRectangle (365,81 80x32), "%.1f", text variable: TEMPERS[1], colour toggle: Nagrev.Auto_IN.1
    RoundedRectangle (249,81 80x32), "%.1f", text variable: Nagrev.T_Actuals[1], colour variable: Nagrev.FillColors[1]
        p3450524324: Nagrev.FrameColors[1]
    Label (192,82 40x32), "T2"
    RoundedRectangle (365,120 80x32), "%.1f", text variable: TEMPERS[2], colour toggle: Nagrev.Auto_IN.2
    RoundedRectangle (249,120 80x32), "%.1f", text variable: Nagrev.T_Actuals[2], colour variable: Nagrev.FillColors[2]
        p3450524324: Nagrev.FrameColors[2]
    Label (192,121 40x32), "T3"
    RoundedRectangle (365,159 80x32), "%.1f", text variable: TEMPERS[3], colour toggle: Nagrev.Auto_IN.3
    RoundedRectangle (249,159 80x32), "%.1f", text variable: Nagrev.T_Actuals[3], colour variable: Nagrev.FillColors[3]
        p3450524324: Nagrev.FrameColors[3]
    Label (192,160 40x32), "T4"
    RoundedRectangle (365,198 80x32), "%.1f", text variable: TEMPERS[4], colour toggle: Nagrev.Auto_IN.4
    RoundedRectangle (249,198 80x32), "%.1f", text variable: Nagrev.T_Actuals[4], colour variable: Nagrev.FillColors[4]
        p3450524324: Nagrev.FrameColors[4]
    Label (192,199 40x32), "T5"
    RoundedRectangle (365,237 80x32), "%.1f", text variable: TEMPERS[5], colour toggle: Nagrev.Auto_IN.5
    RoundedRectangle (249,237 80x32), "%.1f", text variable: Nagrev.T_Actuals[5], colour variable: Nagrev.FillColors[5]
        p3450524324: Nagrev.FrameColors[5]
    Label (192,238 40x32), "T6"
    RoundedRectangle (365,276 80x32), "%.1f", text variable: TEMPERS[6], colour toggle: Nagrev.Auto_IN.6
    RoundedRectangle (249,276 80x32), "%.1f", text variable: Nagrev.T_Actuals[6], colour variable: Nagrev.FillColors[6]
        p3450524324: Nagrev.FrameColors[6]
    Label (192,277 40x32), "T7"
    RoundedRectangle (365,315 80x32), "%.1f", text variable: TEMPERS[7]
    RoundedRectangle (249,315 80x32), "%.1f", text variable: Nagrev.T_Actuals[7], colour variable: Nagrev.FillColors[7]
        p3450524324: Nagrev.FrameColors[7]
    Label (192,316 40x32), "TР"
    RoundedRectangle (365,355 80x32), "%.1f", text variable: REG_W.T_CHIL
    RoundedRectangle (249,355 80x32), "%.1f", text variable: Chiller.T_ACTUAL, colour variable: Chiller.FillColor
        p3450524324: Chiller.FrameColor
    Label (192,356 40x32), "TЧ"
    RoundedRectangle (51,186 30x27), colour toggle: Nagrev.Temper_Reached
    Label (97,186 89x32), "Tемп-ры"
    RoundedRectangle (51,216 30x27), colour toggle: Asda.Pusk
    Label (97,216 89x32), "Головка"
    RoundedRectangle (51,246 30x27), colour toggle: Shnek.Pusk
    Label (97,246 89x32), "Шнек"
    RoundedRectangle (51,276 30x27), colour toggle: Pulling.Pusk
    Label (97,276 89x32), "Тянущее"
    RoundedRectangle (51,6 30x27), colour toggle: Dvp.PVozd_si
    Label (97,6 89x32), "Воздух"
    RoundedRectangle (51,156 30x27), colour toggle: Dvp.Nasos_si
    Label (97,156 89x32), "Насос"
    RoundedRectangle (51,36 30x27), colour toggle: Dvp.Uroven_s_si
    Label (97,36 89x32), "Сырьё"
    RoundedRectangle (51,96 30x27), colour toggle: Dvp.Bunker_si
    Label (97,96 89x32), "Бункер"
    RoundedRectangle (594,12 70x64), colour variable: Chiller.BtnFillColor
        p3450524324: Chiller.BtnFrameColor
    DipSwitch (601,17 58x58), variable: Chiller.Pusk, input disabled if: Chiller.Block, behaviour: TOGGLE, style: Switch-DipSwitch-Gray
    Label (488,21 103x43), "Чиллер и насос"
    Line (599,309) (657,253), invisible if: NOT Shnek.Block
    Line (599,386) (657,330), invisible if: NOT Pulling.Block
    Line (599,230) (657,174), invisible if: NOT Asda.Block
    Line (599,72) (657,16), invisible if: NOT Chiller.Block
    RoundedRectangle (51,126 30x27), colour toggle: Chiller.Connect AND Chiller.Status.0
    Label (97,126 89x32), "Чиллер"
    Button (488,114 80x40), "Режим"
        OnMouseClick: execute { SET_FRAME_INDEX (2); }
    Label (488,88 91x33), "Нагрев"
    Button (488,192 80x40), "Период"
        OnMouseClick: execute { SET_FRAME_INDEX (3); }
    Label (488,166 91x33), "Головка"
    Label (488,245 91x33), "Шнек, %"
    Label (97,307 89x32), "Зажим"
    RoundedRectangle (51,307 30x27), colour toggle: Dvp.Zazh_si
    Label (97,337 46x32), "Нож"
    RoundedRectangle (51,337 30x27), colour toggle: Dvp.Knife_si
    Label (97,367 89x32), "Каретка"
    RoundedRectangle (51,367 30x27), colour toggle: Dvp.Karet_si
    RoundedRectangle (24,306 20x12), colour toggle: Dvp.ZazhIsx_si
    RoundedRectangle (24,320 20x12)
    RoundedRectangle (24,338 20x12), colour toggle: Dvp.KnifeIsx_si
    RoundedRectangle (24,352 20x12), colour toggle: Dvp.KnifeRab_si
    RoundedRectangle (24,369 20x12), colour toggle: Dvp.KarIsx_si
    RoundedRectangle (24,383 20x12), colour toggle: Dvp.KarRab_si
    Label (367,4 96x32), "Уставки"
    Label (227,4 123x32), "Актуальные"
    Line (26,19) (26,289)
    Line (25,19) (44,19)
    Line (26,289) (44,289)
    Button (488,348 80x40), "%.1f", text variable: REG_W.Speed
        OnMouseClick:  Dialog=DlgPulling, Parameters={fSpeed: REG_W.Speed}, Selected={1: }, OpenModal=True, OpenCentered=True
    Label (488,322 91x33), "ТЯУ, %"
    RoundedRectangle (51,66 30x27), colour toggle: Dvp.Uroven_w_si
    Label (97,66 89x32), "Вода"
    Lamp1 (149,337 32x32), variable: Dvp.F_OTR_si, style: Lamp-Lamp1-Red
    Button (488,272 80x40), "%.1f", text variable: REG_W.Qm
        OnMouseClick:  Dialog=DlgTargetRegParams, Parameters={fFreq: REG_W.Freq, fQm: REG_W.Qm, fQm_old: , fSpeed: REG_W.Speed, bQm: , Adapted: }, Selected={1: }, OpenModal=True, OpenCentered=True
END_VISUALIZATION

// Device/Application/Visu/DlgPids
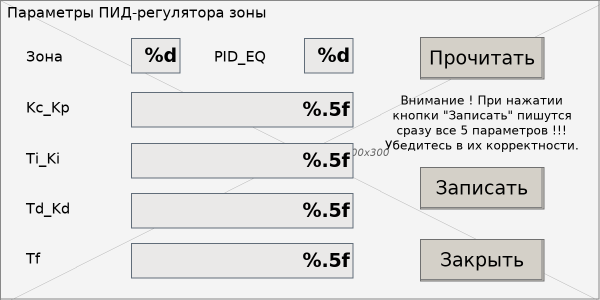
VISUALIZATION DlgPids  // 600x300
VAR_IN_OUT
	bDialogVar	: BOOL;
END_VAR
    Image (0,0 608x305), image: ImagePool.Dialog_win_7_600x300
    Button (420,37 124x42), "Прочитать"
        OnMouseClick: execute { Dvp.pid_read:=TRUE; }
    Button (420,239 124x42), "Закрыть"
        OnMouseClick:  Dialog=DlgPids, Result=OK, NumpadKeypadSet=True
    Label (4,3 296x19), "Параметры ПИД-регулятора зоны"
    Label (23,98 62x19), "Kc_Kp"
    RoundedRectangle (131,92 222x35), "%.5f", text variable: Dvp.Pids[Dvp.pid_index].Kc_Kp
        OnMouseClick: write the text variable via VisuDialogs.Numpad, min 0, max 1000, title "Пропорциональная часть"
    Label (23,149 62x19), "Ti_Ki"
    RoundedRectangle (131,143 222x35), "%.5f", text variable: Dvp.Pids[Dvp.pid_index].Ti_Ki
        OnMouseClick: write the text variable via VisuDialogs.Numpad, min 0, max 1000000, title "Интегральная часть"
    Label (23,199 62x19), "Td_Kd"
    RoundedRectangle (131,193 222x35), "%.5f", text variable: Dvp.Pids[Dvp.pid_index].Td_Kd
        OnMouseClick: write the text variable via VisuDialogs.Numpad, min 0, max 1000, title "Дифференциальная часть"
    RoundedRectangle (131,38 49x35), "%d", text variable: Dvp.zone_index
    Label (23,47 62x19), "Зона"
    Button (420,167 124x42), "Записать"
        OnMouseClick:  Dialog=DlgConfirm, Parameters={bDialogVar: Dvp.pid_write}, Selected={1: }, OpenModal=True, OpenCentered=True
    RoundedRectangle (304,38 49x35), "%d", text variable: Dvp.Pids[Dvp.pid_index].formula
        OnMouseClick: write the text variable via VisuDialogs.Numpad, min 0, max 1, format "Формула ПИД"
    Label (211,47 83x19), "PID_EQ"
    Label (23,249 62x19), "Tf"
    RoundedRectangle (131,243 222x35), "%.5f", text variable: Dvp.Pids[Dvp.pid_index].Tf
        OnMouseClick: write the text variable via VisuDialogs.Numpad, title "Пост.времени дифференцирования"
    Label (389,92 186x79), "Внимание ! При нажатии кнопки "Записать" пишутся сразу все 5 параметров !!! Убедитесь в их корректности."
END_VISUALIZATION

// Device/Application/Visu/VIS_SETTS_1
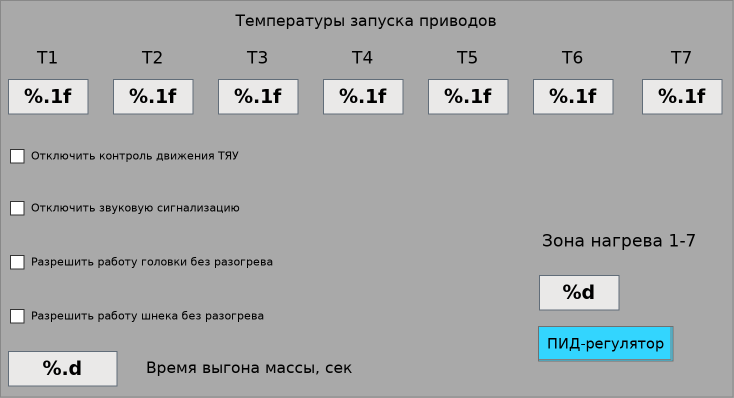
VISUALIZATION VIS_SETTS_1  // 734x398
    Label (219,10 294x28), "Температуры запуска приводов"
    RoundedRectangle (8,79 80x35), "%.1f", text variable: Setts.T_ZAP[0]
        OnMouseClick: write the text variable via VisuDialogs.Numpad, min 160, max 180
    RoundedRectangle (323,79 80x35), "%.1f", text variable: Setts.T_ZAP[3]
        OnMouseClick: write the text variable via VisuDialogs.Numpad, min 300, max 350
    RoundedRectangle (428,79 80x35), "%.1f", text variable: Setts.T_ZAP[4]
        OnMouseClick: write the text variable via VisuDialogs.Numpad, min 220, max 260
    RoundedRectangle (533,79 80x35), "%.1f", text variable: Setts.T_ZAP[5]
        OnMouseClick: write the text variable via VisuDialogs.Numpad, min 230, max 280
    RoundedRectangle (642,79 80x35), "%.1f", text variable: Setts.T_ZAP[6]
        OnMouseClick: write the text variable via VisuDialogs.Numpad, min 230, max 280
    RoundedRectangle (218,79 80x35), "%.1f", text variable: Setts.T_ZAP[2]
        OnMouseClick: write the text variable via VisuDialogs.Numpad, min 300, max 340
    RoundedRectangle (113,79 80x35), "%.1f", text variable: Setts.T_ZAP[1]
        OnMouseClick: write the text variable via VisuDialogs.Numpad, min 310, max 330
    Label (8,46 80x25), "T1"
    Label (113,46 80x25), "T2"
    Label (218,46 80x25), "T3"
    Label (323,46 80x25), "T4"
    Label (428,46 80x25), "T5"
    Label (533,46 80x25), "T6"
    Label (642,46 80x25), "T7"
    Label (539,229 166x28), "Зона нагрева 1-7"
    Button (538,326 135x35), "ПИД-регулятор"
        OnMouseClick:  Dialog=DlgPids, Parameters={bDialogVar: b_dialog}, Selected={1: }, OpenModal=True, OpenCentered=True
    RoundedRectangle (539,275 80x35), "%d", text variable: Dvp.zone_index
        OnMouseClick: write the text variable via VisuDialogs.Numpad, min 1, max 7, title "Введите зону нагрева 1-7"
    Checkbox (8,187 412x42), "Отключить звуковую сигнализацию", variable: Setts.otkl_alarm_zvuk
    Checkbox (8,241 412x42), "Разрешить работу головки без разогрева", variable: Setts.use_servo_without_temp, input disabled if: TRUE
    Checkbox (8,295 412x42), "Разрешить работу шнека без разогрева", variable: Setts.use_shnek_without_temp, input disabled if: TRUE
    Checkbox (8,135 362x42), "Отключить контроль движения ТЯУ", variable: Setts.otkl_c_pulling
    RoundedRectangle (8,351 109x35), "%.d", text variable: TimeVigon
        OnMouseClick: write the text variable via VisuDialogs.Numpad, min 10, max 10000, title "Время выгона массы в сек"
    Label (143,357 294x28), "Время выгона массы, сек"
END_VISUALIZATION

// Device/Application/Visu/VIS_SETTS_3
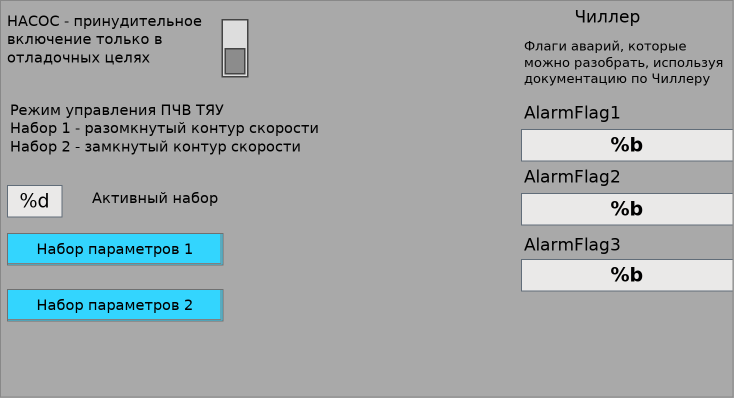
VISUALIZATION VIS_SETTS_3  // 734x398
    RoundedRectangle (521,129 212x32), "%b", text variable: Chiller.AlarmFlag1
    Label (546,5 123x32), "Чиллер"
    Label (521,101 112x32), "AlarmFlag1"
    RoundedRectangle (521,193 212x32), "%b", text variable: Chiller.AlarmFlag2
    Label (521,165 112x32), "AlarmFlag2"
    RoundedRectangle (521,259 212x32), "%b", text variable: Chiller.AlarmFlag3
    Label (521,233 112x32), "AlarmFlag3"
    Label (521,37 209x55), "Флаги аварий, которые можно разобрать, используя документацию по Чиллеру"
    DipSwitch (206,19 58x58), variable: Dvp.Nasos_OTL, behaviour: TOGGLE, style: Switch-DipSwitch-Gray
    Label (4,11 194x77), "НАСОС - принудительное включение только в отладочных целях"
    Label (7,100 315x66), "Режим управления ПЧВ ТЯУ Набор 1 - разомкнутый контур скорости Набор 2 - замкнутый контур скорости"
    Button (7,233 216x32), "Набор параметров 1"
        OnMouseClick: execute {
            PARAM_SET:=1;
            // Запись режима управления тянущего устройства
            // Параметр 1 - Набор данных 1
            // 16#63 - адрес регистра активного набора параметров
            QueuePushReg (ADR (COM2_PRG.WR_REGS), ADR_PULLING, 16#63, ADR (PARAM_SET), 1);
        }
    Button (7,289 216x32), "Набор параметров 2"
        OnMouseClick: execute {
            PARAM_SET:=2;
            // Запись режима управления тянущего устройства
            // Параметр 1 - Набор данных 1
            // 16#63 - адрес регистра активного набора параметров
            QueuePushReg (ADR (COM2_PRG.WR_REGS), ADR_PULLING, 16#63, ADR (PARAM_SET), 1);
        }
    RoundedRectangle (7,185 55x32), "%d", text variable: Pulling.ActiveParamSet
    Label (89,188 134x27), "Активный набор"
END_VISUALIZATION

// Device/Application/Visu/DlgPulling
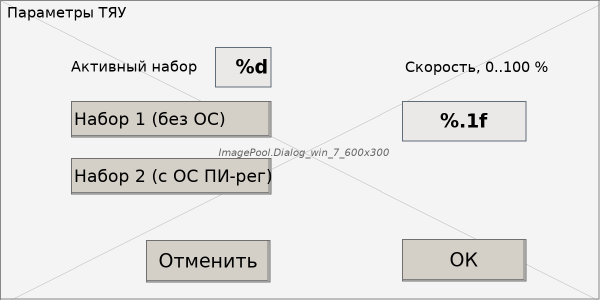
VISUALIZATION DlgPulling  // 600x300
VAR_IN_OUT
	fSpeed	: REAL;
END_VAR
    Image (0,0 608x305), image: ImagePool.Dialog_win_7_600x300
    Button (71,101 200x36), "Набор 1 (без ОС)"
        OnMouseClick: execute {
            PARAM_SET:=1;
            // Запись режима управления тянущего устройства
            // Параметр 1 - Набор данных 1
            // 16#63 - адрес регистра активного набора параметров
            QueuePushReg (ADR (COM2_PRG.WR_REGS), ADR_PULLING, 16#63, ADR (PARAM_SET), 1);
        }
    Button (402,239 124x42), "ОК"
        OnMouseClick:  Dialog=DlgPulling, Result=OK, NumpadKeypadSet=True
    Label (4,3 122x19), "Параметры ТЯУ"
    RoundedRectangle (215,47 56x40), "%d", text variable: Pulling.ActiveParamSet
    Label (68,57 155x19), "Активный набор"
    Button (71,158 200x36), "Набор 2 (с ОС ПИ-рег)"
        OnMouseClick: execute {
            PARAM_SET:=2;
            // Запись режима управления тянущего устройства
            // Параметр 1 - Набор данных 1
            // 16#63 - адрес регистра активного набора параметров
            QueuePushReg (ADR (COM2_PRG.WR_REGS), ADR_PULLING, 16#63, ADR (PARAM_SET), 1);
        }
    Button (146,240 124x42), "Отменить"
        OnMouseClick:  Dialog=DlgPulling, Result=Cancel, NumpadKeypadSet=True
    RoundedRectangle (402,101 124x40), "%.1f", text variable: fSpeed
        OnMouseClick: write the text variable via VisuDialogs.Numpad, min SPEED_MIN, max SPEED_MAX, title "Скорость тянущего, %"
    Label (402,57 147x28), "Скорость, 0..100 %"
END_VISUALIZATION

// Device/Application/Visu/DlgTargetRegParams
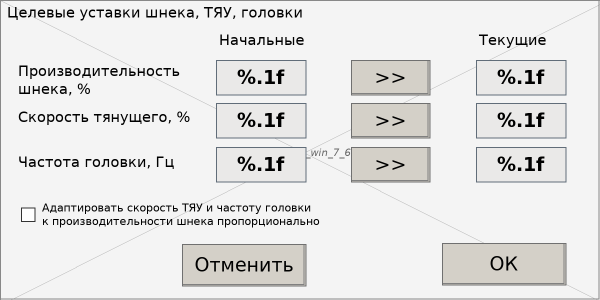
VISUALIZATION DlgTargetRegParams  // 600x300
VAR_IN_OUT
	fQm		: REAL;
	fSpeed	: REAL;
	fFreq	: REAL;
END_VAR

VAR
	fQm_old	: REAL;
	Adapted	: BOOL:=TRUE;
	bQm		: BOOL:=FALSE;
END_VAR
    Image (0,0 608x305), image: ImagePool.Dialog_win_7_600x300
    Button (442,243 124x42), "ОК"
        OnMouseClick:  Dialog=DlgTargetRegParams, Result=OK, NumpadKeypadSet=True
    Label (4,3 341x19), "Целевые уставки шнека, ТЯУ, головки"
    Label (15,62 185x36), "Производительность шнека, %"
    Button (182,244 124x42), "Отменить"
        OnMouseClick:  Dialog=DlgTargetRegParams, Result=Cancel, NumpadKeypadSet=True
    RoundedRectangle (476,103 90x35), "%.1f", text variable: fSpeed
        OnMouseClick: write the text variable via VisuDialogs.Numpad, min SPEED_MIN, max SPEED_MAX, title "Скорость тянущего, %"
    Label (15,107 189x28), "Скорость тянущего, %"
    RoundedRectangle (476,60 90x35), "%.1f", text variable: fQm
        OnMouseClick: write the text variable via VisuDialogs.Numpad, min QM_MIN, max QM_MAX, title "Производительность шнека, %"
        OnMouseClick: execute {
            fQm_old:=fQm; // Производительность
            bQm:=TRUE;
        }
        OnDialogClosed: execute {
            IF bQm THEN
            	IF fQm <> fQm_old THEN
            		IF Adapted AND fQm_old <> 0 THEN
            			fSpeed:=MAX (SPEED_MIN, MIN (SPEED_MAX, fSpeed * fQm / fQm_old));
            			fFreq:=MAX (FREQ_MIN, MIN (FREQ_MAX, fFreq * fQm / fQm_old));
            		END_IF
            		fQm_old:=fQm;
            	END_IF
            	bQm:=FALSE;
            END_IF
        }
    Label (15,152 169x28), "Частота головки, Гц"
    RoundedRectangle (476,147 90x35), "%.1f", text variable: fFreq
        OnMouseClick: write the text variable via VisuDialogs.Numpad, min FREQ_MIN, max FREQ_MAX, title "Частота головки в Гц"
    Checkbox (19,196 393x37), "Адаптировать скорость ТЯУ и частоту головки к производительности шнека пропорционально", variable: Adapted
    RoundedRectangle (216,60 90x35), "%.1f", text variable: REG_W.Qm_b
        OnMouseClick: write the text variable via VisuDialogs.Numpad, min QM_MIN, max QM_MAX, title "Производительность шнека, %"
    RoundedRectangle (216,103 90x35), "%.1f", text variable: REG_W.Speed_b
        OnMouseClick: write the text variable via VisuDialogs.Numpad, min SPEED_MIN, max SPEED_MAX, title "Скорость тянущего, %"
    RoundedRectangle (216,147 90x35), "%.1f", text variable: REG_W.Freq_b
        OnMouseClick: write the text variable via VisuDialogs.Numpad, min FREQ_MIN, max FREQ_MAX, title "Частота головки в Гц"
    Label (216,30 95x28), "Начальные"
    Label (476,30 95x28), "Текущие"
    Button (351,60 79x35), ">>"
        OnMouseClick: execute {
            fQm:=REG_W.Qm_b;
            IF Adapted THEN
            	fSpeed:=REG_W.Speed_b;
            	fFreq:=REG_W.Freq_b;
            END_IF
        }
    Button (351,103 79x35), ">>"
        OnMouseClick: execute { fSpeed:=REG_W.Speed_b; }
    Button (351,147 79x35), ">>"
        OnMouseClick: execute { fFreq:=REG_W.Freq_b; }
END_VISUALIZATION

(* text list AsdaTextList (id | default)
  0 | Ожидание команды
  1 | Инициализация сервопривода
  2 | Поиск реперной точки (Homing)
  3 | Формирование каркаса
  4 | Операция отладочного перемещения
  5 | Операция задержки
  6 | Включение сервопривода
  7 | Экстренный останов
  8 | Отключение сервопривода
  9 | Установка параметров сервопривода
  10 | Обработка ошибки
  11 | Перемещение в реперную точку
  12 | Ожидание соединения
   |  *)

(* text list AG_DVP (id | default)
  9 | Нулевая скорость движения заготовки
  8 | Каретка в крайнем положении
  7 | Превышено время возврата каретки на исходный концевик
  6 | Превышено время схода каретки с исходного концевика
  5 | Превышено время движения ножа
  4 | Превышено время схода ножа с исходного концевика
  3 | Превышено время движения зажима
  2 | Нож не на исходном концевике
  1 | Зажим не на исходном концевике
  0 | Каретка не на исходном концевике
   |  *)

(* text list DvpTextList (id | default)
  0 | Система в исходном состоянии
  1 | Система в режиме РАЗОГРЕВ
  2 | Система в рабочем состоянии
  3 | Система в режиме выгона массы
   |  *)

(* text list AG_CONNECT (id | default)
  4 | Нет соединения с Чиллером
  3 | Нет соединения с ПЧВ тянущего устройства
  2 | Нет соединения с ПЧВ шнека
  1 | Нет соединения с контроллером DVP
  0 | Нет соединение с сервоприводом ASDA-A2
   |  *)

(* text list MSGS (id | default)
  13 | Низкий уровень воды в баке !!!
  12 | Перегрев ПЧВ тянущего устройства
  11 | Перегрузка по току ПЧВ тянущего устройства
  10 | Напряжение не в норме ПЧВ тянущего устройства
  9 | Предупреждение от ПЧВ тянущего устройства
  8 | Перегрев ПЧВ шнека
  7 | Перегрузка по току ПЧВ шнека
  6 | Напряжение не в норме ПЧВ шнека
  5 | Предупреждение от ПЧВ шнека
  4 | Низкое давление воздуха !!!
  3 | Низкий уровень сырья в бункере !!!
  2 | Выведите бункер !!!
  1 | Бункер выведен !!!
  0 | Система вышла на режим !
   |  *)

(* text list AG_AVAR (id | default)
  4 | 
  3 | Низкая температура одной из зон
  2 | Превышена температура одной из зон
  1 | Температура одной из зон ниже температуры запуска привода
  0 | Превышена критическая температура одной из зон
   |  *)

(* text list AG_DEV (id | default)
  11 | Тестовая авария
  13 | Авария Чиллера
  10 | Аварийный сигнал ПЧВ тянущего устройства
  7 | Аварийный сигнал ПЧВ шнека
  6 | Тестовая ошибка
  5 | Превышено время операции отладки
  4 | РЕЗЕРВ АВАРИИ
  3 | Превышено время операции HOMING
  2 | Ошибка инициализации Р2-30 или Р3-06
  1 | Сигнал предупреждения от сервопривода
  0 | Сигнал аварии от сервопривода
   |  *)

(* text list AG_CHILLER (id | default)
  35 | Авария Чиллера
  34 | Неисправен датчик элетрического сопротивления жидкости в Чиллере
  33 | Повышение элетрического удельного сопротивления жидкости в Чиллере
  32 | Обнаружена утечка воды Чиллера
  31 | Обнаружен сигнал контакта входа 2 Чиллера
  30 | Обнаружен сигнал контакта входа 1 Чиллера
  29 | Обслуживание компрессора двигателя Чиллера
  28 | Обслуживание вентилятора двигателя Чиллера
  27 | Обслуживание насоса Чиллера
  26 | Неисправность датчика давления на входе компрессора Чиллера
  25 | Неисправность датчика давления нагнетания компрессора Чиллера
  24 | Неисправность датчика давления нагнетания Чиллера
  23 | Неисправность датчика температуры на входе компрессора Чиллера
  22 | Неисправность датчика температуры на входе Чиллера
  21 | Неисправность датчика температуры на выходе Чиллера
  20 | Сработал предохранитель постоянного тока в Чиллере
  19 | Ошибка памяти контроллера Чиллера
  18 | Ошибка связи с контроллером Чиллера
  17 | Перегрузка компрессора Чиллера
  16 | Падение давления на низкой стороне контура хладагента Чиллера
  15 | Повышение давления на низкой стороне контура хладагента Чиллера
  14 | Падение давления на высокой стороне контура хладагента Чиллера
  13 | Unused
  12 | Высокое давление нагнетания компрессора Чиллера
  11 | Низкая температура нагревания Чиллера
  10 | Низкая температура на входе компрессора Чиллера
  9 | Высокая температура на входе компрессора Чиллера
  8 | Падение давления нагнетания Чиллера
  7 | Повышение давления нагнетания Чиллера
  6 | Ненормальная работа насоса Чиллера
  5 | Высокая давление нагнетания Чиллера
  4 | Высокая температура воды на входе Чиллера
  3 | Температура на выходе Чиллера...
  2 | Температура на выходе Чиллера выросла
  1 | Высокая температура воды на выходе Чиллера
  0 | Низкий уровень воды в Чиллере
   |  *)
